LIN {X 0,Y 390.04,Z 157.401,A -85,B 0,C 180,E1 -11467.551,E2 -11467.551} C_VEL
LIN {X 0,Y 390.051,Z 157.369,A -85,B 0,C 180,E1 -11470.821,E2 -11470.821} C_VEL
LIN {X 0,Y 390.052,Z 157.382,A -85,B 0,C 180,E1 -11473.887,E2 -11473.887} C_VEL
LIN {X 0,Y 390.054,Z 157.401,A -85,B 0,C 180,E1 -11476.79,E2 -11476.79} C_VEL
LIN {X 0,Y 390.051,Z 157.386,A -85,B 0,C 180,E1 -11479.561,E2 -11479.561} C_VEL
LIN {X 0,Y 390.041,Z 157.403,A -85,B 0,C 180,E1 -11482.449,E2 -11482.449} C_VEL
LIN {X 0,Y 390.063,Z 157.38,A -85,B 0,C 180,E1 -11485.976,E2 -11485.976} C_VEL
LIN {X 0,Y 390.046,Z 157.398,A -85,B 0,C 180,E1 -11489.868,E2 -11489.868} C_VEL
LIN {X 0,Y 390.109,Z 157.374,A -85,B 0,C 180,E1 -11493.232,E2 -11493.232} C_VEL
LIN {X 0,Y 390.102,Z 157.391,A -85,B 0,C 180,E1 -11496.751,E2 -11496.751} C_VEL
LIN {X 0,Y 390.099,Z 157.374,A -85,B 0,C 180,E1 -11499.983,E2 -11499.983} C_VEL
LIN {X 0,Y 390.134,Z 157.379,A -85,B 0,C 180,E1 -11503.249,E2 -11503.249} C_VEL
LIN {X 0,Y 390.19,Z 157.377,A -85,B 0,C 180,E1 -11506.562,E2 -11506.562} C_VEL
LIN {X 0,Y 390.201,Z 157.357,A -85,B 0,C 180,E1 -11510.672,E2 -11510.672} C_VEL
LIN {X 0,Y 390.315,Z 157.357,A -85,B 0,C 180,E1 -11512.76,E2 -11512.76} C_VEL
LIN {X 0,Y 390.224,Z 157.374,A -85,B 0,C 180,E1 -11514.834,E2 -11514.834} C_VEL
LIN {X 0,Y 390.417,Z 157.337,A -85,B 0,C 180,E1 -11517.937,E2 -11517.937} C_VEL
LIN {X 0,Y 390.544,Z 157.311,A -85,B 0,C 180,E1 -11520.001,E2 -11520.001} C_VEL
LIN {X 0,Y 390.308,Z 157.36,A -85,B 0,C 180,E1 -11523.097,E2 -11523.097} C_VEL
LIN {X 0,Y 390.326,Z 157.359,A -85,B 0,C 180,E1 -11526.202,E2 -11526.202} C_VEL
LIN {X 0,Y 390.202,Z 157.354,A -85,B 0,C 180,E1 -11529.329,E2 -11529.329} C_VEL
LIN {X 0,Y 390.192,Z 157.381,A -85,B 0,C 180,E1 -11533.439,E2 -11533.439} C_VEL
LIN {X 0,Y 390.147,Z 157.369,A -85,B 0,C 180,E1 -11537.308,E2 -11537.308} C_VEL
LIN {X 0,Y 390.086,Z 157.38,A -85,B 0,C 180,E1 -11540.471,E2 -11540.471} C_VEL
LIN {X 0,Y 390.088,Z 157.392,A -85,B 0,C 180,E1 -11543.351,E2 -11543.351} C_VEL
LIN {X 0,Y 390.112,Z 157.373,A -85,B 0,C 180,E1 -11546.769,E2 -11546.769} C_VEL
LIN {X 0,Y 390.038,Z 157.398,A -85,B 0,C 180,E1 -11550.3,E2 -11550.3} C_VEL
LIN {X 0,Y 390.067,Z 157.381,A -85,B 0,C 180,E1 -11554.025,E2 -11554.025} C_VEL
LIN {X 0,Y 390.041,Z 157.398,A -85,B 0,C 180,E1 -11557.551,E2 -11557.551} C_VEL
LIN {X 0,Y 390.056,Z 157.392,A -85,B 0,C 180,E1 -11560.822,E2 -11560.822} C_VEL
LIN {X 0,Y 390.054,Z 157.396,A -85,B 0,C 180,E1 -11563.887,E2 -11563.887} C_VEL
LIN {X 0,Y 390.058,Z 157.398,A -85,B 0,C 180,E1 -11566.79,E2 -11566.79} C_VEL
LIN {X 0,Y 390.057,Z 157.377,A -85,B 0,C 180,E1 -11569.561,E2 -11569.561} C_VEL
LIN {X 0,Y 390.046,Z 157.401,A -85,B 0,C 180,E1 -11572.45,E2 -11572.45} C_VEL
LIN {X 0,Y 390.07,Z 157.396,A -85,B 0,C 180,E1 -11575.976,E2 -11575.976} C_VEL
LIN {X 0,Y 390.108,Z 157.507,A -85,B 0,C 180,E1 -11579.707,E2 -11579.707} C_VEL
LIN {X 0,Y 392.073,Z 167.322,A -85,B 0,C 180,E1 -11582.801,E2 -11582.801} C_VEL
LIN {X 0,Y 392.8,Z 173.578,A -85,B 0,C 180,E1 -11584.57,E2 -11584.57} C_VEL
LIN {X 0,Y 391.761,Z 185.813,A -85,B 0,C 180,E1 -11587.869,E2 -11587.869} C_VEL
LIN {X 0,Y 391.287,Z 191.653,A -85,B 0,C 180,E1 -11589.464,E2 -11589.464} C_VEL
LIN {X 0,Y 391.844,Z 194.823,A -85,B 0,C 180,E1 -11589.615,E2 -11589.615} C_VEL
LIN {X 0,Y 396.817,Z 222.018,A -85,B 0,C 180,E1 -11590.391,E2 -11590.391} C_VEL
LIN {X 0,Y 395.833,Z 296.555,A -85,B 0,C 180,E1 -11591.764,E2 -11591.764} C_VEL
LIN {X 0,Y 395.429,Z 307.324,A -85,B 0,C 180,E1 -11592.08,E2 -11592.08} C_VEL
LIN {X 0,Y 394.95,Z 316.424,A -85,B 0,C 180,E1 -11592.459,E2 -11592.459} C_VEL
LIN {X 0,Y 394.344,Z 326.787,A -85,B 0,C 180,E1 -11593.032,E2 -11593.032} C_VEL
LIN {X 0,Y 393.605,Z 335.919,A -85,B 0,C 180,E1 -11593.667,E2 -11593.667} C_VEL
LIN {X 0,Y 392.878,Z 344.915,A -85,B 0,C 180,E1 -11594.435,E2 -11594.435} C_VEL
LIN {X 0,Y 392.118,Z 353.643,A -85,B 0,C 180,E1 -11595.335,E2 -11595.335} C_VEL
LIN {X 0,Y 391.462,Z 361.4,A -85,B 0,C 180,E1 -11596.288,E2 -11596.288} C_VEL
LIN {X 0,Y 390.904,Z 368.261,A -85,B 0,C 180,E1 -11597.277,E2 -11597.277} C_VEL
LIN {X 0,Y 390.301,Z 374.462,A -85,B 0,C 180,E1 -11598.313,E2 -11598.313} C_VEL
LIN {X 0,Y 389.761,Z 381,A -85,B 0,C 180,E1 -11599.612,E2 -11599.612} C_VEL
LIN {X 0,Y 389.383,Z 385.501,A -85,B 0,C 180,E1 -11600.651,E2 -11600.651} C_VEL
LIN {X 0,Y 389.017,Z 390.993,A -85,B 0,C 180,E1 -11602.213,E2 -11602.213} C_VEL
LIN {X 0,Y 388.797,Z 395.317,A -85,B 0,C 180,E1 -11603.774,E2 -11603.774} C_VEL
LIN {X 0,Y 388.74,Z 397.684,A -85,B 0,C 180,E1 -11604.814,E2 -11604.814} C_VEL
LIN {X 0,Y 388.7,Z 399.482,A -85,B 0,C 180,E1 -11605.853,E2 -11605.853} C_VEL
LIN {X 0,Y 388.661,Z 401.926,A -85,B 0,C 180,E1 -11607.927,E2 -11607.927} C_VEL
LIN {X 0,Y 388.704,Z 402.515,A -85,B 0,C 180,E1 -11608.964,E2 -11608.964} C_VEL
LIN {X 0,Y 388.704,Z 402.515,A -85,B 0,C 180,E1 -11611.036,E2 -11611.036} C_VEL
LIN {X 0,Y 388.661,Z 401.926,A -85,B 0,C 180,E1 -11612.073,E2 -11612.073} C_VEL
LIN {X 0,Y 388.7,Z 399.482,A -85,B 0,C 180,E1 -11614.147,E2 -11614.147} C_VEL
LIN {X 0,Y 388.726,Z 396.43,A -85,B 0,C 180,E1 -11615.751,E2 -11615.751} C_VEL
LIN {X 0,Y 388.933,Z 392.546,A -85,B 0,C 180,E1 -11617.267,E2 -11617.267} C_VEL
LIN {X 0,Y 389.251,Z 387.417,A -85,B 0,C 180,E1 -11618.828,E2 -11618.828} C_VEL
LIN {X 0,Y 389.651,Z 382.155,A -85,B 0,C 180,E1 -11620.128,E2 -11620.128} C_VEL
LIN {X 0,Y 390.156,Z 375.837,A -85,B 0,C 180,E1 -11621.428,E2 -11621.428} C_VEL
LIN {X 0,Y 390.745,Z 369.888,A -85,B 0,C 180,E1 -11622.464,E2 -11622.464} C_VEL
LIN {X 0,Y 391.32,Z 362.959,A -85,B 0,C 180,E1 -11623.502,E2 -11623.502} C_VEL
LIN {X 0,Y 392.026,Z 354.778,A -85,B 0,C 180,E1 -11624.536,E2 -11624.536} C_VEL
LIN {X 0,Y 392.733,Z 346.266,A -85,B 0,C 180,E1 -11625.437,E2 -11625.437} C_VEL
LIN {X 0,Y 393.454,Z 337.55,A -85,B 0,C 180,E1 -11626.206,E2 -11626.206} C_VEL
LIN {X 0,Y 394.214,Z 327.793,A -85,B 0,C 180,E1 -11626.907,E2 -11626.907} C_VEL
LIN {X 0,Y 394.887,Z 317.712,A -85,B 0,C 180,E1 -11627.477,E2 -11627.477} C_VEL
LIN {X 0,Y 395.36,Z 308.197,A -85,B 0,C 180,E1 -11627.89,E2 -11627.89} C_VEL
LIN {X 0,Y 395.814,Z 297.888,A -85,B 0,C 180,E1 -11628.203,E2 -11628.203} C_VEL
LIN {X 0,Y 396.74,Z 227.164,A -85,B 0,C 180,E1 -11629.517,E2 -11629.517} C_VEL
LIN {X 0,Y 396.668,Z 221.21,A -85,B 0,C 180,E1 -11629.632,E2 -11629.632} C_VEL
LIN {X 0,Y 391.483,Z 193.035,A -85,B 0,C 180,E1 -11630.439,E2 -11630.439} C_VEL
LIN {X 0,Y 391.316,Z 191.446,A -85,B 0,C 180,E1 -11630.569,E2 -11630.569} C_VEL
LIN {X 0,Y 392.571,Z 176.893,A -85,B 0,C 180,E1 -11634.597,E2 -11634.597} C_VEL
LIN {X 0,Y 392.857,Z 172.015,A -85,B 0,C 180,E1 -11635.94,E2 -11635.94} C_VEL
LIN {X 0,Y 391.366,Z 163.735,A -85,B 0,C 180,E1 -11638.366,E2 -11638.366} C_VEL
LIN {X 0,Y 390.098,Z 157.409,A -85,B 0,C 180,E1 -11640.369,E2 -11640.369} C_VEL
LIN {X 0,Y 390.07,Z 157.397,A -85,B 0,C 180,E1 -11644.024,E2 -11644.024} C_VEL
LIN {X 0,Y 390.046,Z 157.401,A -85,B 0,C 180,E1 -11647.55,E2 -11647.55} C_VEL
LIN {X 0,Y 390.057,Z 157.379,A -85,B 0,C 180,E1 -11650.821,E2 -11650.821} C_VEL
LIN {X 0,Y 390.055,Z 157.398,A -85,B 0,C 180,E1 -11653.885,E2 -11653.885} C_VEL
LIN {X 0,Y 390.057,Z 157.396,A -85,B 0,C 180,E1 -11656.789,E2 -11656.789} C_VEL
LIN {X 0,Y 390.056,Z 157.389,A -85,B 0,C 180,E1 -11659.56,E2 -11659.56} C_VEL
LIN {X 0,Y 390.041,Z 157.398,A -85,B 0,C 180,E1 -11662.449,E2 -11662.449} C_VEL
LIN {X 0,Y 390.067,Z 157.381,A -85,B 0,C 180,E1 -11665.975,E2 -11665.975} C_VEL
LIN {X 0,Y 390.045,Z 157.396,A -85,B 0,C 180,E1 -11669.868,E2 -11669.868} C_VEL
LIN {X 0,Y 390.112,Z 157.373,A -85,B 0,C 180,E1 -11673.231,E2 -11673.231} C_VEL
LIN {X 0,Y 390.105,Z 157.391,A -85,B 0,C 180,E1 -11676.75,E2 -11676.75} C_VEL
LIN {X 0,Y 390.102,Z 157.377,A -85,B 0,C 180,E1 -11679.982,E2 -11679.982} C_VEL
LIN {X 0,Y 390.136,Z 157.379,A -85,B 0,C 180,E1 -11683.248,E2 -11683.248} C_VEL
LIN {X 0,Y 390.192,Z 157.381,A -85,B 0,C 180,E1 -11686.561,E2 -11686.561} C_VEL
LIN {X 0,Y 390.202,Z 157.354,A -85,B 0,C 180,E1 -11690.671,E2 -11690.671} C_VEL
LIN {X 0,Y 390.326,Z 157.359,A -85,B 0,C 180,E1 -11693.798,E2 -11693.798} C_VEL
LIN {X 0,Y 390.415,Z 157.346,A -85,B 0,C 180,E1 -11697.936,E2 -11697.936} C_VEL
LIN {X 0,Y 390.544,Z 157.311,A -85,B 0,C 180,E1 -11699.999,E2 -11699.999} C_VEL
LIN {X 0,Y 390.312,Z 157.36,A -85,B 0,C 180,E1 -11703.096,E2 -11703.096} C_VEL
LIN {X 0,Y 390.306,Z 157.361,A -85,B 0,C 180,E1 -11706.625,E2 -11706.625} C_VEL
LIN {X 0,Y 390.201,Z 157.357,A -85,B 0,C 180,E1 -11709.328,E2 -11709.328} C_VEL
LIN {X 0,Y 390.19,Z 157.377,A -85,B 0,C 180,E1 -11713.438,E2 -11713.438} C_VEL
LIN {X 0,Y 390.144,Z 157.379,A -85,B 0,C 180,E1 -11717.307,E2 -11717.307} C_VEL
LIN {X 0,Y 390.083,Z 157.384,A -85,B 0,C 180,E1 -11720.47,E2 -11720.47} C_VEL
LIN {X 0,Y 390.085,Z 157.394,A -85,B 0,C 180,E1 -11723.35,E2 -11723.35} C_VEL
LIN {X 0,Y 390.109,Z 157.374,A -85,B 0,C 180,E1 -11726.768,E2 -11726.768} C_VEL
LIN {X 0,Y 390.038,Z 157.399,A -85,B 0,C 180,E1 -11730.299,E2 -11730.299} C_VEL
LIN {X 0,Y 390.063,Z 157.38,A -85,B 0,C 180,E1 -11734.024,E2 -11734.024} C_VEL
LIN {X 0,Y 390.041,Z 157.403,A -85,B 0,C 180,E1 -11737.551,E2 -11737.551} C_VEL
LIN {X 0,Y 390.052,Z 157.386,A -85,B 0,C 180,E1 -11740.821,E2 -11740.821} C_VEL
LIN {X 0,Y 390.052,Z 157.396,A -85,B 0,C 180,E1 -11743.886,E2 -11743.886} C_VEL
LIN {X 0,Y 390.054,Z 157.368,A -85,B 0,C 180,E1 -11746.79,E2 -11746.79} C_VEL
LIN {X 0,Y 390.051,Z 157.377,A -85,B 0,C 180,E1 -11749.56,E2 -11749.56} C_VEL
LIN {X 0,Y 390.04,Z 157.401,A -85,B 0,C 180,E1 -11752.449,E2 -11752.449} C_VEL
LIN {X 0,Y 390.063,Z 157.376,A -85,B 0,C 180,E1 -11755.975,E2 -11755.975} C_VEL
LIN {X 0,Y 390.045,Z 157.402,A -85,B 0,C 180,E1 -11758.498,E2 -11758.498} C_VEL
LIN {X 0,Y 390.113,Z 157.387,A -85,B 0,C 180,E1 -11762.07,E2 -11762.07} C_VEL
LIN {X 0,Y 390.076,Z 157.396,A -85,B 0,C 180,E1 -11765.519,E2 -11765.519} C_VEL
LIN {X 0,Y 390.052,Z 157.401,A -85,B 0,C 180,E1 -11768.878,E2 -11768.878} C_VEL
LIN {X 0,Y 390.124,Z 157.392,A -85,B 0,C 180,E1 -11772.167,E2 -11772.167} C_VEL
LIN {X 0,Y 390.14,Z 157.389,A -85,B 0,C 180,E1 -11775.393,E2 -11775.393} C_VEL
LIN {X 0,Y 390.145,Z 157.389,A -85,B 0,C 180,E1 -11778.571,E2 -11778.571} C_VEL
LIN {X 0,Y 390.382,Z 157.657,A -85,B 0,C 180,E1 -11781.829,E2 -11781.829} C_VEL
LIN {X 0,Y 390.711,Z 158.919,A -85,B 0,C 180,E1 -11782.459,E2 -11782.459} C_VEL
LIN {X 0,Y 392.085,Z 161.236,A -85,B 0,C 180,E1 -11783.568,E2 -11783.568} C_VEL
LIN {X 0,Y 394.112,Z 162.919,A -85,B 0,C 180,E1 -11785.397,E2 -11785.397} C_VEL
LIN {X 0,Y 395.582,Z 163.492,A -85,B 0,C 180,E1 -11787.454,E2 -11787.454} C_VEL
LIN {X 0,Y 396.128,Z 163.931,A -85,B 0,C 180,E1 -11788.983,E2 -11788.983} C_VEL
LIN {X 0,Y 396.323,Z 163.848,A -85,B 0,C 180,E1 -11790,E2 -11790} C_VEL
LIN {X 0,Y 396.07,Z 163.803,A -85,B 0,C 180,E1 -11791.525,E2 -11791.525} C_VEL
LIN {X 0,Y 395.354,Z 163.371,A -85,B 0,C 180,E1 -11793.057,E2 -11793.057} C_VEL
LIN {X 0,Y 393.693,Z 162.658,A -85,B 0,C 180,E1 -11794.992,E2 -11794.992} C_VEL
LIN {X 0,Y 391.897,Z 161.019,A -85,B 0,C 180,E1 -11796.565,E2 -11796.565} C_VEL
LIN {X 0,Y 390.579,Z 158.502,A -85,B 0,C 180,E1 -11797.684,E2 -11797.684} C_VEL
LIN {X 0,Y 390.341,Z 157.593,A -85,B 0,C 180,E1 -11798.281,E2 -11798.281} C_VEL
LIN {X 0,Y 390.145,Z 157.389,A -85,B 0,C 180,E1 -11801.429,E2 -11801.429} C_VEL
LIN {X 0,Y 390.14,Z 157.39,A -85,B 0,C 180,E1 -11804.607,E2 -11804.607} C_VEL
LIN {X 0,Y 390.124,Z 157.392,A -85,B 0,C 180,E1 -11807.833,E2 -11807.833} C_VEL
LIN {X 0,Y 390.052,Z 157.401,A -85,B 0,C 180,E1 -11811.122,E2 -11811.122} C_VEL
LIN {X 0,Y 390.076,Z 157.396,A -85,B 0,C 180,E1 -11814.481,E2 -11814.481} C_VEL
LIN {X 0,Y 390.111,Z 157.387,A -85,B 0,C 180,E1 -11818.025,E2 -11818.025} C_VEL
LIN {X 0,Y 390.022,Z 157.396,A -85,B 0,C 180,E1 -11820.799,E2 -11820.799} C_VEL
LIN {X 0,Y 389.356,Z 157.487,A -85,B 0,C 180,E1 -11821.661,E2 -11821.661} C_VEL
LIN {X 0,Y 386.503,Z 157.831,A -85,B 0,C 180,E1 -11823.063,E2 -11823.063} C_VEL
LIN {X 0,Y 384.095,Z 158.119,A -85,B 0,C 180,E1 -11824.195,E2 -11824.195} C_VEL
LIN {X 0,Y 383.071,Z 158.245,A -85,B 0,C 180,E1 -11825.071,E2 -11825.071} C_VEL
LIN {X 0,Y 382.994,Z 158.257,A -85,B 0,C 180,E1 -11825.368,E2 -11825.368} C_VEL
LIN {X 0,Y 383.001,Z 158.279,A -85,B 0,C 180,E1 -11828.601,E2 -11828.601} C_VEL
LIN {X 0,Y 382.978,Z 158.243,A -85,B 0,C 180,E1 -11831.348,E2 -11831.348} C_VEL
LIN {X 0,Y 382.994,Z 158.262,A -85,B 0,C 180,E1 -11834.304,E2 -11834.304} C_VEL
LIN {X 0,Y 383.005,Z 158.274,A -85,B 0,C 180,E1 -11837.24,E2 -11837.24} C_VEL
LIN {X 0,Y 383.011,Z 158.267,A -85,B 0,C 180,E1 -11840.414,E2 -11840.414} C_VEL
LIN {X 0,Y 383.022,Z 158.271,A -85,B 0,C 180,E1 -11844.045,E2 -11844.045} C_VEL
LIN {X 0,Y 382.983,Z 158.274,A -85,B 0,C 180,E1 -11847.578,E2 -11847.578} C_VEL
LIN {X 0,Y 382.992,Z 158.275,A -85,B 0,C 180,E1 -11850.301,E2 -11850.301} C_VEL
LIN {X 0,Y 383.052,Z 158.251,A -85,B 0,C 180,E1 -11852.698,E2 -11852.698} C_VEL
LIN {X 0,Y 383.048,Z 158.266,A -85,B 0,C 180,E1 -11855.04,E2 -11855.04} C_VEL
LIN {X 0,Y 382.989,Z 158.271,A -85,B 0,C 180,E1 -11858.469,E2 -11858.469} C_VEL
LIN {X 0,Y 383.058,Z 158.247,A -85,B 0,C 180,E1 -11861.827,E2 -11861.827} C_VEL
LIN {X 0,Y 383.106,Z 158.261,A -85,B 0,C 180,E1 -11865.119,E2 -11865.119} C_VEL
LIN {X 0,Y 383.093,Z 158.249,A -85,B 0,C 180,E1 -11868.358,E2 -11868.358} C_VEL
LIN {X 0,Y 383.3,Z 158.225,A -85,B 0,C 180,E1 -11871.933,E2 -11871.933} C_VEL
LIN {X 0,Y 383.196,Z 158.25,A -85,B 0,C 180,E1 -11874.739,E2 -11874.739} C_VEL
LIN {X 0,Y 383.384,Z 158.213,A -85,B 0,C 180,E1 -11877.899,E2 -11877.899} C_VEL
LIN {X 0,Y 383.514,Z 158.186,A -85,B 0,C 180,E1 -11880.001,E2 -11880.001} C_VEL
LIN {X 0,Y 383.244,Z 158.24,A -85,B 0,C 180,E1 -11883.154,E2 -11883.154} C_VEL
LIN {X 0,Y 383.282,Z 158.236,A -85,B 0,C 180,E1 -11886.317,E2 -11886.317} C_VEL
LIN {X 0,Y 383.148,Z 158.231,A -85,B 0,C 180,E1 -11889.503,E2 -11889.503} C_VEL
LIN {X 0,Y 383.123,Z 158.261,A -85,B 0,C 180,E1 -11893.537,E2 -11893.537} C_VEL
LIN {X 0,Y 383.092,Z 158.245,A -85,B 0,C 180,E1 -11897.455,E2 -11897.455} C_VEL
LIN {X 0,Y 383.029,Z 158.26,A -85,B 0,C 180,E1 -11900.649,E2 -11900.649} C_VEL
LIN {X 0,Y 383.032,Z 158.268,A -85,B 0,C 180,E1 -11903.808,E2 -11903.808} C_VEL
LIN {X 0,Y 383.055,Z 158.252,A -85,B 0,C 180,E1 -11907.303,E2 -11907.303} C_VEL
LIN {X 0,Y 382.982,Z 158.281,A -85,B 0,C 180,E1 -11910.919,E2 -11910.919} C_VEL
LIN {X 0,Y 383.017,Z 158.26,A -85,B 0,C 180,E1 -11914.669,E2 -11914.669} C_VEL
LIN {X 0,Y 382.997,Z 158.276,A -85,B 0,C 180,E1 -11917.904,E2 -11917.904} C_VEL
LIN {X 0,Y 382.983,Z 158.275,A -85,B 0,C 180,E1 -11921.348,E2 -11921.348} C_VEL
LIN {X 0,Y 382.996,Z 158.273,A -85,B 0,C 180,E1 -11924.304,E2 -11924.304} C_VEL
LIN {X 0,Y 383.011,Z 158.274,A -85,B 0,C 180,E1 -11927.241,E2 -11927.241} C_VEL
LIN {X 0,Y 383.017,Z 158.257,A -85,B 0,C 180,E1 -11930.414,E2 -11930.414} C_VEL
LIN {X 0,Y 383.027,Z 158.262,A -85,B 0,C 180,E1 -11934.045,E2 -11934.045} C_VEL
LIN {X 0,Y 382.988,Z 158.271,A -85,B 0,C 180,E1 -11937.579,E2 -11937.579} C_VEL
LIN {X 0,Y 383.085,Z 158.439,A -85,B 0,C 180,E1 -11939.428,E2 -11939.428} C_VEL
LIN {X 0,Y 385.219,Z 169.231,A -85,B 0,C 180,E1 -11942.864,E2 -11942.864} C_VEL
LIN {X 0,Y 385.823,Z 174.445,A -85,B 0,C 180,E1 -11944.366,E2 -11944.366} C_VEL
LIN {X 0,Y 384.863,Z 185.625,A -85,B 0,C 180,E1 -11947.451,E2 -11947.451} C_VEL
LIN {X 0,Y 384.402,Z 191.46,A -85,B 0,C 180,E1 -11949.078,E2 -11949.078} C_VEL
LIN {X 0,Y 384.807,Z 194.101,A -85,B 0,C 180,E1 -11949.215,E2 -11949.215} C_VEL
LIN {X 0,Y 389.909,Z 221.418,A -85,B 0,C 180,E1 -11950.021,E2 -11950.021} C_VEL
LIN {X 0,Y 390.122,Z 228.726,A -85,B 0,C 180,E1 -11950.172,E2 -11950.172} C_VEL
LIN {X 0,Y 389.1,Z 296.364,A -85,B 0,C 180,E1 -11951.437,E2 -11951.437} C_VEL
LIN {X 0,Y 388.692,Z 307.133,A -85,B 0,C 180,E1 -11951.758,E2 -11951.758} C_VEL
LIN {X 0,Y 388.187,Z 316.232,A -85,B 0,C 180,E1 -11952.143,E2 -11952.143} C_VEL
LIN {X 0,Y 387.553,Z 326.595,A -85,B 0,C 180,E1 -11952.726,E2 -11952.726} C_VEL
LIN {X 0,Y 386.785,Z 335.727,A -85,B 0,C 180,E1 -11953.371,E2 -11953.371} C_VEL
LIN {X 0,Y 386.013,Z 344.723,A -85,B 0,C 180,E1 -11954.151,E2 -11954.151} C_VEL
LIN {X 0,Y 385.217,Z 353.451,A -85,B 0,C 180,E1 -11955.067,E2 -11955.067} C_VEL
LIN {X 0,Y 384.53,Z 361.407,A -85,B 0,C 180,E1 -11956.064,E2 -11956.064} C_VEL
LIN {X 0,Y 383.793,Z 369.696,A -85,B 0,C 180,E1 -11957.306,E2 -11957.306} C_VEL
LIN {X 0,Y 383.174,Z 375.645,A -85,B 0,C 180,E1 -11958.36,E2 -11958.36} C_VEL
LIN {X 0,Y 382.642,Z 381.963,A -85,B 0,C 180,E1 -11959.684,E2 -11959.684} C_VEL
LIN {X 0,Y 382.207,Z 387.225,A -85,B 0,C 180,E1 -11961.008,E2 -11961.008} C_VEL
LIN {X 0,Y 381.861,Z 392.354,A -85,B 0,C 180,E1 -11962.598,E2 -11962.598} C_VEL
LIN {X 0,Y 381.688,Z 395.641,A -85,B 0,C 180,E1 -11963.883,E2 -11963.883} C_VEL
LIN {X 0,Y 381.641,Z 397.491,A -85,B 0,C 180,E1 -11964.717,E2 -11964.717} C_VEL
LIN {X 0,Y 381.625,Z 399.291,A -85,B 0,C 180,E1 -11965.776,E2 -11965.776} C_VEL
LIN {X 0,Y 381.56,Z 401.734,A -85,B 0,C 180,E1 -11967.889,E2 -11967.889} C_VEL
LIN {X 0,Y 381.604,Z 402.323,A -85,B 0,C 180,E1 -11968.945,E2 -11968.945} C_VEL
LIN {X 0,Y 381.604,Z 402.323,A -85,B 0,C 180,E1 -11971.055,E2 -11971.055} C_VEL
LIN {X 0,Y 381.56,Z 401.734,A -85,B 0,C 180,E1 -11972.111,E2 -11972.111} C_VEL
LIN {X 0,Y 381.625,Z 399.291,A -85,B 0,C 180,E1 -11974.224,E2 -11974.224} C_VEL
LIN {X 0,Y 381.64,Z 397.491,A -85,B 0,C 180,E1 -11975.283,E2 -11975.283} C_VEL
LIN {X 0,Y 381.781,Z 393.884,A -85,B 0,C 180,E1 -11976.872,E2 -11976.872} C_VEL
LIN {X 0,Y 382.058,Z 389.14,A -85,B 0,C 180,E1 -11978.462,E2 -11978.462} C_VEL
LIN {X 0,Y 382.525,Z 383.118,A -85,B 0,C 180,E1 -11980.052,E2 -11980.052} C_VEL
LIN {X 0,Y 383.053,Z 377.021,A -85,B 0,C 180,E1 -11981.375,E2 -11981.375} C_VEL
LIN {X 0,Y 383.643,Z 371.322,A -85,B 0,C 180,E1 -11982.43,E2 -11982.43} C_VEL
LIN {X 0,Y 384.369,Z 362.766,A -85,B 0,C 180,E1 -11983.751,E2 -11983.751} C_VEL
LIN {X 0,Y 385.145,Z 354.586,A -85,B 0,C 180,E1 -11984.801,E2 -11984.801} C_VEL
LIN {X 0,Y 385.892,Z 346.074,A -85,B 0,C 180,E1 -11985.718,E2 -11985.718} C_VEL
LIN {X 0,Y 386.646,Z 337.359,A -85,B 0,C 180,E1 -11986.5,E2 -11986.5} C_VEL
LIN {X 0,Y 387.424,Z 327.601,A -85,B 0,C 180,E1 -11987.212,E2 -11987.212} C_VEL
LIN {X 0,Y 388.107,Z 317.52,A -85,B 0,C 180,E1 -11987.793,E2 -11987.793} C_VEL
LIN {X 0,Y 388.626,Z 308.006,A -85,B 0,C 180,E1 -11988.211,E2 -11988.211} C_VEL
LIN {X 0,Y 389.083,Z 297.696,A -85,B 0,C 180,E1 -11988.529,E2 -11988.529} C_VEL
LIN {X 0,Y 390.038,Z 230.896,A -85,B 0,C 180,E1 -11989.791,E2 -11989.791} C_VEL
LIN {X 0,Y 389.98,Z 222.068,A -85,B 0,C 180,E1 -11989.963,E2 -11989.963} C_VEL
LIN {X 0,Y 384.819,Z 193.984,A -85,B 0,C 180,E1 -11990.787,E2 -11990.787} C_VEL
LIN {X 0,Y 384.39,Z 191.454,A -85,B 0,C 180,E1 -11990.923,E2 -11990.923} C_VEL
LIN {X 0,Y 385.748,Z 176.712,A -85,B 0,C 180,E1 -11995.061,E2 -11995.061} C_VEL
LIN {X 0,Y 385.917,Z 173.701,A -85,B 0,C 180,E1 -11995.917,E2 -11995.917} C_VEL
LIN {X 0,Y 384.497,Z 165.445,A -85,B 0,C 180,E1 -11998.375,E2 -11998.375} C_VEL
LIN {X 0,Y 383.049,Z 158.304,A -85,B 0,C 180,E1 -12000.653,E2 -12000.653} C_VEL
LIN {X 0,Y 383.019,Z 158.268,A -85,B 0,C 180,E1 -12004.667,E2 -12004.667} C_VEL
LIN {X 0,Y 383.002,Z 158.277,A -85,B 0,C 180,E1 -12007.903,E2 -12007.903} C_VEL
LIN {X 0,Y 382.984,Z 158.263,A -85,B 0,C 180,E1 -12011.347,E2 -12011.347} C_VEL
LIN {X 0,Y 382.996,Z 158.274,A -85,B 0,C 180,E1 -12014.303,E2 -12014.303} C_VEL
LIN {X 0,Y 383.01,Z 158.277,A -85,B 0,C 180,E1 -12017.24,E2 -12017.24} C_VEL
LIN {X 0,Y 383.013,Z 158.265,A -85,B 0,C 180,E1 -12020.413,E2 -12020.413} C_VEL
LIN {X 0,Y 383.024,Z 158.267,A -85,B 0,C 180,E1 -12024.044,E2 -12024.044} C_VEL
LIN {X 0,Y 382.986,Z 158.275,A -85,B 0,C 180,E1 -12027.577,E2 -12027.577} C_VEL
LIN {X 0,Y 382.991,Z 158.275,A -85,B 0,C 180,E1 -12030.299,E2 -12030.299} C_VEL
LIN {X 0,Y 383.079,Z 158.252,A -85,B 0,C 180,E1 -12034.02,E2 -12034.02} C_VEL
LIN {X 0,Y 383.011,Z 158.273,A -85,B 0,C 180,E1 -12037.335,E2 -12037.335} C_VEL
LIN {X 0,Y 383.058,Z 158.247,A -85,B 0,C 180,E1 -12040.716,E2 -12040.716} C_VEL
LIN {X 0,Y 383.078,Z 158.258,A -85,B 0,C 180,E1 -12044.026,E2 -12044.026} C_VEL
LIN {X 0,Y 383.134,Z 158.252,A -85,B 0,C 180,E1 -12047.283,E2 -12047.283} C_VEL
LIN {X 0,Y 383.148,Z 158.231,A -85,B 0,C 180,E1 -12050.497,E2 -12050.497} C_VEL
LIN {X 0,Y 383.282,Z 158.236,A -85,B 0,C 180,E1 -12053.683,E2 -12053.683} C_VEL
LIN {X 0,Y 383.382,Z 158.222,A -85,B 0,C 180,E1 -12057.898,E2 -12057.898} C_VEL
LIN {X 0,Y 383.514,Z 158.186,A -85,B 0,C 180,E1 -12059.999,E2 -12059.999} C_VEL
LIN {X 0,Y 383.248,Z 158.239,A -85,B 0,C 180,E1 -12063.153,E2 -12063.153} C_VEL
LIN {X 0,Y 383.266,Z 158.238,A -85,B 0,C 180,E1 -12066.618,E2 -12066.618} C_VEL
LIN {X 0,Y 383.256,Z 158.225,A -85,B 0,C 180,E1 -12068.435,E2 -12068.435} C_VEL
LIN {X 0,Y 383.093,Z 158.249,A -85,B 0,C 180,E1 -12071.642,E2 -12071.642} C_VEL
LIN {X 0,Y 383.106,Z 158.261,A -85,B 0,C 180,E1 -12074.881,E2 -12074.881} C_VEL
LIN {X 0,Y 383.058,Z 158.247,A -85,B 0,C 180,E1 -12078.173,E2 -12078.173} C_VEL
LIN {X 0,Y 382.989,Z 158.271,A -85,B 0,C 180,E1 -12081.531,E2 -12081.531} C_VEL
LIN {X 0,Y 383.048,Z 158.266,A -85,B 0,C 180,E1 -12084.96,E2 -12084.96} C_VEL
LIN {X 0,Y 383.044,Z 158.261,A -85,B 0,C 180,E1 -12088.492,E2 -12088.492} C_VEL
LIN {X 0,Y 383.006,Z 158.272,A -85,B 0,C 180,E1 -12092.149,E2 -12092.149} C_VEL
LIN {X 0,Y 383.013,Z 158.256,A -85,B 0,C 180,E1 -12094.668,E2 -12094.668} C_VEL
LIN {X 0,Y 382.997,Z 158.277,A -85,B 0,C 180,E1 -12097.904,E2 -12097.904} C_VEL
LIN {X 0,Y 382.98,Z 158.27,A -85,B 0,C 180,E1 -12101.347,E2 -12101.347} C_VEL
LIN {X 0,Y 382.994,Z 158.274,A -85,B 0,C 180,E1 -12104.304,E2 -12104.304} C_VEL
LIN {X 0,Y 383.005,Z 158.239,A -85,B 0,C 180,E1 -12107.24,E2 -12107.24} C_VEL
LIN {X 0,Y 383.01,Z 158.266,A -85,B 0,C 180,E1 -12110.413,E2 -12110.413} C_VEL
LIN {X 0,Y 383.022,Z 158.262,A -85,B 0,C 180,E1 -12114.045,E2 -12114.045} C_VEL
LIN {X 0,Y 383.033,Z 158.272,A -85,B 0,C 180,E1 -12117.853,E2 -12117.853} C_VEL
LIN {X 0,Y 383.059,Z 158.261,A -85,B 0,C 180,E1 -12121.72,E2 -12121.72} C_VEL
LIN {X 0,Y 383.048,Z 158.273,A -85,B 0,C 180,E1 -12125.04,E2 -12125.04} C_VEL
LIN {X 0,Y 382.989,Z 158.281,A -85,B 0,C 180,E1 -12128.469,E2 -12128.469} C_VEL
LIN {X 0,Y 383.085,Z 158.268,A -85,B 0,C 180,E1 -12131.828,E2 -12131.828} C_VEL
LIN {X 0,Y 383.106,Z 158.266,A -85,B 0,C 180,E1 -12135.118,E2 -12135.118} C_VEL
LIN {X 0,Y 383.113,Z 158.39,A -85,B 0,C 180,E1 -12138.359,E2 -12138.359} C_VEL
LIN {X 0,Y 383.303,Z 159.256,A -85,B 0,C 180,E1 -12138.867,E2 -12138.867} C_VEL
LIN {X 0,Y 384.444,Z 161.599,A -85,B 0,C 180,E1 -12139.533,E2 -12139.533} C_VEL
LIN {X 0,Y 386.582,Z 163.495,A -85,B 0,C 180,E1 -12140.583,E2 -12140.583} C_VEL
LIN {X 0,Y 388.921,Z 164.829,A -85,B 0,C 180,E1 -12141.896,E2 -12141.896} C_VEL
LIN {X 0,Y 390.34,Z 167.396,A -85,B 0,C 180,E1 -12142.955,E2 -12142.955} C_VEL
LIN {X 0,Y 391.933,Z 169.071,A -85,B 0,C 180,E1 -12144.211,E2 -12144.211} C_VEL
LIN {X 0,Y 393.437,Z 170.033,A -85,B 0,C 180,E1 -12145.646,E2 -12145.646} C_VEL
LIN {X 0,Y 394.719,Z 170.512,A -85,B 0,C 180,E1 -12147.449,E2 -12147.449} C_VEL
LIN {X 0,Y 395.266,Z 170.977,A -85,B 0,C 180,E1 -12148.981,E2 -12148.981} C_VEL
LIN {X 0,Y 395.458,Z 170.896,A -85,B 0,C 180,E1 -12150,E2 -12150} C_VEL
LIN {X 0,Y 395.202,Z 170.852,A -85,B 0,C 180,E1 -12151.529,E2 -12151.529} C_VEL
LIN {X 0,Y 394.244,Z 170.355,A -85,B 0,C 180,E1 -12153.368,E2 -12153.368} C_VEL
LIN {X 0,Y 392.65,Z 169.62,A -85,B 0,C 180,E1 -12155.134,E2 -12155.134} C_VEL
LIN {X 0,Y 390.787,Z 167.978,A -85,B 0,C 180,E1 -12156.713,E2 -12156.713} C_VEL
LIN {X 0,Y 389.246,Z 165.411,A -85,B 0,C 180,E1 -12157.901,E2 -12157.901} C_VEL
LIN {X 0,Y 388.306,Z 164.316,A -85,B 0,C 180,E1 -12158.456,E2 -12158.456} C_VEL
LIN {X 0,Y 385.837,Z 163.007,A -85,B 0,C 180,E1 -12159.766,E2 -12159.766} C_VEL
LIN {X 0,Y 383.934,Z 160.79,A -85,B 0,C 180,E1 -12160.748,E2 -12160.748} C_VEL
LIN {X 0,Y 383.222,Z 158.963,A -85,B 0,C 180,E1 -12161.236,E2 -12161.236} C_VEL
LIN {X 0,Y 383.115,Z 158.297,A -85,B 0,C 180,E1 -12161.91,E2 -12161.91} C_VEL
LIN {X 0,Y 383.106,Z 158.266,A -85,B 0,C 180,E1 -12164.882,E2 -12164.882} C_VEL
LIN {X 0,Y 383.085,Z 158.268,A -85,B 0,C 180,E1 -12168.172,E2 -12168.172} C_VEL
LIN {X 0,Y 382.989,Z 158.281,A -85,B 0,C 180,E1 -12171.531,E2 -12171.531} C_VEL
LIN {X 0,Y 383.048,Z 158.273,A -85,B 0,C 180,E1 -12174.96,E2 -12174.96} C_VEL
LIN {X 0,Y 383.045,Z 158.26,A -85,B 0,C 180,E1 -12178.492,E2 -12178.492} C_VEL
LIN {X 0,Y 383.023,Z 158.274,A -85,B 0,C 180,E1 -12182.432,E2 -12182.432} C_VEL
LIN {X 0,Y 382.994,Z 158.257,A -85,B 0,C 180,E1 -12185.368,E2 -12185.368} C_VEL
LIN {X 0,Y 382.357,Z 158.348,A -85,B 0,C 180,E1 -12186.246,E2 -12186.246} C_VEL
LIN {X 0,Y 379.562,Z 158.711,A -85,B 0,C 180,E1 -12187.674,E2 -12187.674} C_VEL
LIN {X 0,Y 377.157,Z 159.01,A -85,B 0,C 180,E1 -12188.828,E2 -12188.828} C_VEL
LIN {X 0,Y 376.086,Z 159.131,A -85,B 0,C 180,E1 -12189.72,E2 -12189.72} C_VEL
LIN {X 0,Y 375.978,Z 159.137,A -85,B 0,C 180,E1 -12190.022,E2 -12190.022} C_VEL
LIN {X 0,Y 375.927,Z 159.136,A -85,B 0,C 180,E1 -12193.766,E2 -12193.766} C_VEL
LIN {X 0,Y 375.93,Z 159.16,A -85,B 0,C 180,E1 -12196.811,E2 -12196.811} C_VEL
LIN {X 0,Y 375.959,Z 159.146,A -85,B 0,C 180,E1 -12200.538,E2 -12200.538} C_VEL
LIN {X 0,Y 375.96,Z 159.15,A -85,B 0,C 180,E1 -12203.496,E2 -12203.496} C_VEL
LIN {X 0,Y 375.955,Z 159.136,A -85,B 0,C 180,E1 -12205.889,E2 -12205.889} C_VEL
LIN {X 0,Y 375.963,Z 159.152,A -85,B 0,C 180,E1 -12209.688,E2 -12209.688} C_VEL
LIN {X 0,Y 375.997,Z 159.132,A -85,B 0,C 180,E1 -12212.142,E2 -12212.142} C_VEL
LIN {X 0,Y 376.002,Z 159.141,A -85,B 0,C 180,E1 -12214.539,E2 -12214.539} C_VEL
LIN {X 0,Y 375.959,Z 159.152,A -85,B 0,C 180,E1 -12218.046,E2 -12218.046} C_VEL
LIN {X 0,Y 376.004,Z 159.122,A -85,B 0,C 180,E1 -12221.474,E2 -12221.474} C_VEL
LIN {X 0,Y 376.054,Z 159.14,A -85,B 0,C 180,E1 -12224.833,E2 -12224.833} C_VEL
LIN {X 0,Y 376.045,Z 159.129,A -85,B 0,C 180,E1 -12228.137,E2 -12228.137} C_VEL
LIN {X 0,Y 376.254,Z 159.101,A -85,B 0,C 180,E1 -12231.878,E2 -12231.878} C_VEL
LIN {X 0,Y 376.168,Z 159.125,A -85,B 0,C 180,E1 -12234.64,E2 -12234.64} C_VEL
LIN {X 0,Y 376.35,Z 159.089,A -85,B 0,C 180,E1 -12237.86,E2 -12237.86} C_VEL
LIN {X 0,Y 376.483,Z 159.061,A -85,B 0,C 180,E1 -12240.001,E2 -12240.001} C_VEL
LIN {X 0,Y 376.183,Z 159.121,A -85,B 0,C 180,E1 -12243.214,E2 -12243.214} C_VEL
LIN {X 0,Y 376.24,Z 159.113,A -85,B 0,C 180,E1 -12246.436,E2 -12246.436} C_VEL
LIN {X 0,Y 376.116,Z 159.106,A -85,B 0,C 180,E1 -12249.682,E2 -12249.682} C_VEL
LIN {X 0,Y 376.087,Z 159.136,A -85,B 0,C 180,E1 -12253.658,E2 -12253.658} C_VEL
LIN {X 0,Y 376.041,Z 159.121,A -85,B 0,C 180,E1 -12257.607,E2 -12257.607} C_VEL
LIN {X 0,Y 375.976,Z 159.14,A -85,B 0,C 180,E1 -12260.833,E2 -12260.833} C_VEL
LIN {X 0,Y 375.992,Z 159.145,A -85,B 0,C 180,E1 -12264.282,E2 -12264.282} C_VEL
LIN {X 0,Y 376.018,Z 159.127,A -85,B 0,C 180,E1 -12266.653,E2 -12266.653} C_VEL
LIN {X 0,Y 375.964,Z 159.152,A -85,B 0,C 180,E1 -12270.313,E2 -12270.313} C_VEL
LIN {X 0,Y 375.959,Z 159.137,A -85,B 0,C 180,E1 -12274.112,E2 -12274.112} C_VEL
LIN {X 0,Y 375.952,Z 159.156,A -85,B 0,C 180,E1 -12276.742,E2 -12276.742} C_VEL
LIN {X 0,Y 375.987,Z 159.14,A -85,B 0,C 180,E1 -12279.971,E2 -12279.971} C_VEL
LIN {X 0,Y 375.93,Z 159.155,A -85,B 0,C 180,E1 -12283.767,E2 -12283.767} C_VEL
LIN {X 0,Y 375.935,Z 159.157,A -85,B 0,C 180,E1 -12286.811,E2 -12286.811} C_VEL
LIN {X 0,Y 375.964,Z 159.136,A -85,B 0,C 180,E1 -12290.538,E2 -12290.538} C_VEL
LIN {X 0,Y 375.966,Z 159.147,A -85,B 0,C 180,E1 -12293.496,E2 -12293.496} C_VEL
LIN {X 0,Y 375.962,Z 159.152,A -85,B 0,C 180,E1 -12295.889,E2 -12295.889} C_VEL
LIN {X 0,Y 375.988,Z 159.295,A -85,B 0,C 180,E1 -12299.095,E2 -12299.095} C_VEL
LIN {X 0,Y 377.978,Z 169.05,A -85,B 0,C 180,E1 -12302.3,E2 -12302.3} C_VEL
LIN {X 0,Y 378.867,Z 175.313,A -85,B 0,C 180,E1 -12304.156,E2 -12304.156} C_VEL
LIN {X 0,Y 377.992,Z 185.438,A -85,B 0,C 180,E1 -12307.018,E2 -12307.018} C_VEL
LIN {X 0,Y 377.482,Z 191.342,A -85,B 0,C 180,E1 -12308.688,E2 -12308.688} C_VEL
LIN {X 0,Y 378.456,Z 196.459,A -85,B 0,C 180,E1 -12308.9,E2 -12308.9} C_VEL
LIN {X 0,Y 383.326,Z 222.881,A -85,B 0,C 180,E1 -12309.695,E2 -12309.695} C_VEL
LIN {X 0,Y 383.032,Z 254.972,A -85,B 0,C 180,E1 -12310.305,E2 -12310.305} C_VEL
LIN {X 0,Y 382.334,Z 297.504,A -85,B 0,C 180,E1 -12311.131,E2 -12311.131} C_VEL
LIN {X 0,Y 381.921,Z 307.815,A -85,B 0,C 180,E1 -12311.458,E2 -12311.458} C_VEL
LIN {X 0,Y 381.355,Z 317.328,A -85,B 0,C 180,E1 -12311.881,E2 -12311.881} C_VEL
LIN {X 0,Y 380.707,Z 327.411,A -85,B 0,C 180,E1 -12312.474,E2 -12312.474} C_VEL
LIN {X 0,Y 379.85,Z 337.167,A -85,B 0,C 180,E1 -12313.196,E2 -12313.196} C_VEL
LIN {X 0,Y 378.925,Z 347.234,A -85,B 0,C 180,E1 -12314.123,E2 -12314.123} C_VEL
LIN {X 0,Y 377.876,Z 358.621,A -85,B 0,C 180,E1 -12315.442,E2 -12315.442} C_VEL
LIN {X 0,Y 377.032,Z 367.877,A -85,B 0,C 180,E1 -12316.801,E2 -12316.801} C_VEL
LIN {X 0,Y 376.374,Z 374.078,A -85,B 0,C 180,E1 -12317.874,E2 -12317.874} C_VEL
LIN {X 0,Y 375.696,Z 380.614,A -85,B 0,C 180,E1 -12319.219,E2 -12319.219} C_VEL
LIN {X 0,Y 375.324,Z 385.116,A -85,B 0,C 180,E1 -12320.298,E2 -12320.298} C_VEL
LIN {X 0,Y 374.882,Z 390.607,A -85,B 0,C 180,E1 -12321.917,E2 -12321.917} C_VEL
LIN {X 0,Y 374.633,Z 394.932,A -85,B 0,C 180,E1 -12323.537,E2 -12323.537} C_VEL
LIN {X 0,Y 374.551,Z 397.299,A -85,B 0,C 180,E1 -12324.617,E2 -12324.617} C_VEL
LIN {X 0,Y 374.529,Z 399.099,A -85,B 0,C 180,E1 -12325.695,E2 -12325.695} C_VEL
LIN {X 0,Y 374.459,Z 401.542,A -85,B 0,C 180,E1 -12327.849,E2 -12327.849} C_VEL
LIN {X 0,Y 374.504,Z 402.132,A -85,B 0,C 180,E1 -12328.925,E2 -12328.925} C_VEL
LIN {X 0,Y 374.504,Z 402.132,A -85,B 0,C 180,E1 -12331.075,E2 -12331.075} C_VEL
LIN {X 0,Y 374.459,Z 401.542,A -85,B 0,C 180,E1 -12332.151,E2 -12332.151} C_VEL
LIN {X 0,Y 374.529,Z 399.098,A -85,B 0,C 180,E1 -12334.305,E2 -12334.305} C_VEL
LIN {X 0,Y 374.583,Z 395.831,A -85,B 0,C 180,E1 -12336.064,E2 -12336.064} C_VEL
LIN {X 0,Y 374.794,Z 392.162,A -85,B 0,C 180,E1 -12337.542,E2 -12337.542} C_VEL
LIN {X 0,Y 375.163,Z 387.032,A -85,B 0,C 180,E1 -12339.162,E2 -12339.162} C_VEL
LIN {X 0,Y 375.626,Z 381.77,A -85,B 0,C 180,E1 -12340.511,E2 -12340.511} C_VEL
LIN {X 0,Y 376.203,Z 375.453,A -85,B 0,C 180,E1 -12341.858,E2 -12341.858} C_VEL
LIN {X 0,Y 376.864,Z 369.504,A -85,B 0,C 180,E1 -12342.931,E2 -12342.931} C_VEL
LIN {X 0,Y 377.596,Z 361.36,A -85,B 0,C 180,E1 -12344.176,E2 -12344.176} C_VEL
LIN {X 0,Y 378.496,Z 352.125,A -85,B 0,C 180,E1 -12345.343,E2 -12345.343} C_VEL
LIN {X 0,Y 379.437,Z 341.828,A -85,B 0,C 180,E1 -12346.407,E2 -12346.407} C_VEL
LIN {X 0,Y 380.5,Z 329.423,A -85,B 0,C 180,E1 -12347.397,E2 -12347.397} C_VEL
LIN {X 0,Y 381.298,Z 318.617,A -85,B 0,C 180,E1 -12348.052,E2 -12348.052} C_VEL
LIN {X 0,Y 381.847,Z 308.689,A -85,B 0,C 180,E1 -12348.511,E2 -12348.511} C_VEL
LIN {X 0,Y 382.337,Z 298.837,A -85,B 0,C 180,E1 -12348.834,E2 -12348.834} C_VEL
LIN {X 0,Y 382.804,Z 274.614,A -85,B 0,C 180,E1 -12349.324,E2 -12349.324} C_VEL
LIN {X 0,Y 383.354,Z 223.195,A -85,B 0,C 180,E1 -12350.297,E2 -12350.297} C_VEL
LIN {X 0,Y 378.048,Z 194.446,A -85,B 0,C 180,E1 -12351.164,E2 -12351.164} C_VEL
LIN {X 0,Y 377.471,Z 191.356,A -85,B 0,C 180,E1 -12351.308,E2 -12351.308} C_VEL
LIN {X 0,Y 378.946,Z 176.531,A -85,B 0,C 180,E1 -12355.543,E2 -12355.543} C_VEL
LIN {X 0,Y 378.518,Z 171.762,A -85,B 0,C 180,E1 -12356.972,E2 -12356.972} C_VEL
LIN {X 0,Y 376.396,Z 161.131,A -85,B 0,C 180,E1 -12360.274,E2 -12360.274} C_VEL
LIN {X 0,Y 375.977,Z 159.205,A -85,B 0,C 180,E1 -12360.965,E2 -12360.965} C_VEL
LIN {X 0,Y 375.981,Z 159.144,A -85,B 0,C 180,E1 -12364.667,E2 -12364.667} C_VEL
LIN {X 0,Y 375.977,Z 159.149,A -85,B 0,C 180,E1 -12368.27,E2 -12368.27} C_VEL
LIN {X 0,Y 375.935,Z 159.144,A -85,B 0,C 180,E1 -12371.6,E2 -12371.6} C_VEL
LIN {X 0,Y 375.927,Z 159.152,A -85,B 0,C 180,E1 -12375.268,E2 -12375.268} C_VEL
LIN {X 0,Y 375.934,Z 159.154,A -85,B 0,C 180,E1 -12378.399,E2 -12378.399} C_VEL
LIN {X 0,Y 375.972,Z 159.153,A -85,B 0,C 180,E1 -12381.729,E2 -12381.729} C_VEL
LIN {X 0,Y 375.979,Z 159.137,A -85,B 0,C 180,E1 -12385.332,E2 -12385.332} C_VEL
LIN {X 0,Y 375.957,Z 159.151,A -85,B 0,C 180,E1 -12388.437,E2 -12388.437} C_VEL
LIN {X 0,Y 375.982,Z 159.136,A -85,B 0,C 180,E1 -12392.14,E2 -12392.14} C_VEL
LIN {X 0,Y 376.005,Z 159.134,A -85,B 0,C 180,E1 -12394.538,E2 -12394.538} C_VEL
LIN {X 0,Y 375.966,Z 159.148,A -85,B 0,C 180,E1 -12398.045,E2 -12398.045} C_VEL
LIN {X 0,Y 376.007,Z 159.122,A -85,B 0,C 180,E1 -12401.473,E2 -12401.473} C_VEL
LIN {X 0,Y 376.056,Z 159.14,A -85,B 0,C 180,E1 -12404.832,E2 -12404.832} C_VEL
LIN {X 0,Y 376.047,Z 159.134,A -85,B 0,C 180,E1 -12408.136,E2 -12408.136} C_VEL
LIN {X 0,Y 376.218,Z 159.103,A -85,B 0,C 180,E1 -12411.917,E2 -12411.917} C_VEL
LIN {X 0,Y 376.168,Z 159.13,A -85,B 0,C 180,E1 -12414.639,E2 -12414.639} C_VEL
LIN {X 0,Y 376.348,Z 159.098,A -85,B 0,C 180,E1 -12417.859,E2 -12417.859} C_VEL
LIN {X 0,Y 376.483,Z 159.061,A -85,B 0,C 180,E1 -12419.999,E2 -12419.999} C_VEL
LIN {X 0,Y 376.186,Z 159.119,A -85,B 0,C 180,E1 -12423.212,E2 -12423.212} C_VEL
LIN {X 0,Y 376.231,Z 159.114,A -85,B 0,C 180,E1 -12426.609,E2 -12426.609} C_VEL
LIN {X 0,Y 376.202,Z 159.102,A -85,B 0,C 180,E1 -12428.595,E2 -12428.595} C_VEL
LIN {X 0,Y 376.045,Z 159.129,A -85,B 0,C 180,E1 -12431.863,E2 -12431.863} C_VEL
LIN {X 0,Y 376.054,Z 159.14,A -85,B 0,C 180,E1 -12435.167,E2 -12435.167} C_VEL
LIN {X 0,Y 376.004,Z 159.122,A -85,B 0,C 180,E1 -12438.526,E2 -12438.526} C_VEL
LIN {X 0,Y 375.959,Z 159.152,A -85,B 0,C 180,E1 -12441.954,E2 -12441.954} C_VEL
LIN {X 0,Y 376.002,Z 159.141,A -85,B 0,C 180,E1 -12445.461,E2 -12445.461} C_VEL
LIN {X 0,Y 375.971,Z 159.143,A -85,B 0,C 180,E1 -12449.078,E2 -12449.078} C_VEL
LIN {X 0,Y 375.945,Z 159.152,A -85,B 0,C 180,E1 -12452.828,E2 -12452.828} C_VEL
LIN {X 0,Y 375.953,Z 159.141,A -85,B 0,C 180,E1 -12455.415,E2 -12455.415} C_VEL
LIN {X 0,Y 375.971,Z 159.151,A -85,B 0,C 180,E1 -12458.271,E2 -12458.271} C_VEL
LIN {X 0,Y 375.93,Z 159.151,A -85,B 0,C 180,E1 -12461.601,E2 -12461.601} C_VEL
LIN {X 0,Y 375.95,Z 159.143,A -85,B 0,C 180,E1 -12465.264,E2 -12465.264} C_VEL
LIN {X 0,Y 375.935,Z 159.125,A -85,B 0,C 180,E1 -12469.133,E2 -12469.133} C_VEL
LIN {X 0,Y 375.961,Z 159.153,A -85,B 0,C 180,E1 -12471.912,E2 -12471.912} C_VEL
LIN {X 0,Y 375.975,Z 159.127,A -85,B 0,C 180,E1 -12475.333,E2 -12475.333} C_VEL
LIN {X 0,Y 375.973,Z 159.154,A -85,B 0,C 180,E1 -12478.44,E2 -12478.44} C_VEL
LIN {X 0,Y 375.998,Z 159.146,A -85,B 0,C 180,E1 -12482.142,E2 -12482.142} C_VEL
LIN {X 0,Y 376.002,Z 159.151,A -85,B 0,C 180,E1 -12484.539,E2 -12484.539} C_VEL
LIN {X 0,Y 375.959,Z 159.156,A -85,B 0,C 180,E1 -12488.046,E2 -12488.046} C_VEL
LIN {X 0,Y 376.02,Z 159.149,A -85,B 0,C 180,E1 -12491.474,E2 -12491.474} C_VEL
LIN {X 0,Y 376.054,Z 159.144,A -85,B 0,C 180,E1 -12494.833,E2 -12494.833} C_VEL
LIN {X 0,Y 376.115,Z 159.431,A -85,B 0,C 180,E1 -12496.109,E2 -12496.109} C_VEL
LIN {X 0,Y 376.404,Z 160.523,A -85,B 0,C 180,E1 -12496.467,E2 -12496.467} C_VEL
LIN {X 0,Y 377.861,Z 163.024,A -85,B 0,C 180,E1 -12497.103,E2 -12497.103} C_VEL
LIN {X 0,Y 380.043,Z 164.683,A -85,B 0,C 180,E1 -12497.945,E2 -12497.945} C_VEL
LIN {X 0,Y 381.205,Z 165.432,A -85,B 0,C 180,E1 -12498.434,E2 -12498.434} C_VEL
LIN {X 0,Y 382.765,Z 167.993,A -85,B 0,C 180,E1 -12499.152,E2 -12499.152} C_VEL
LIN {X 0,Y 385.027,Z 170.222,A -85,B 0,C 180,E1 -12500.287,E2 -12500.287} C_VEL
LIN {X 0,Y 387.591,Z 171.68,A -85,B 0,C 180,E1 -12501.659,E2 -12501.659} C_VEL
LIN {X 0,Y 389.285,Z 174.435,A -85,B 0,C 180,E1 -12502.841,E2 -12502.841} C_VEL
LIN {X 0,Y 391.041,Z 176.14,A -85,B 0,C 180,E1 -12504.198,E2 -12504.198} C_VEL
LIN {X 0,Y 392.756,Z 177.219,A -85,B 0,C 180,E1 -12505.896,E2 -12505.896} C_VEL
LIN {X 0,Y 393.915,Z 177.6,A -85,B 0,C 180,E1 -12507.579,E2 -12507.579} C_VEL
LIN {X 0,Y 394.407,Z 178.003,A -85,B 0,C 180,E1 -12508.979,E2 -12508.979} C_VEL
LIN {X 0,Y 394.593,Z 177.943,A -85,B 0,C 180,E1 -12510,E2 -12510} C_VEL
LIN {X 0,Y 394.096,Z 177.716,A -85,B 0,C 180,E1 -12512.044,E2 -12512.044} C_VEL
LIN {X 0,Y 393.066,Z 177.319,A -85,B 0,C 180,E1 -12513.725,E2 -12513.725} C_VEL
LIN {X 0,Y 391.609,Z 176.583,A -85,B 0,C 180,E1 -12515.277,E2 -12515.277} C_VEL
LIN {X 0,Y 389.867,Z 175.113,A -85,B 0,C 180,E1 -12516.729,E2 -12516.729} C_VEL
LIN {X 0,Y 388.033,Z 172.482,A -85,B 0,C 180,E1 -12518.061,E2 -12518.061} C_VEL
LIN {X 0,Y 387.368,Z 171.385,A -85,B 0,C 180,E1 -12518.477,E2 -12518.477} C_VEL
LIN {X 0,Y 384.676,Z 169.97,A -85,B 0,C 180,E1 -12519.88,E2 -12519.88} C_VEL
LIN {X 0,Y 382.443,Z 167.627,A -85,B 0,C 180,E1 -12520.991,E2 -12520.991} C_VEL
LIN {X 0,Y 380.868,Z 165.114,A -85,B 0,C 180,E1 -12521.711,E2 -12521.711} C_VEL
LIN {X 0,Y 378.262,Z 163.429,A -85,B 0,C 180,E1 -12522.746,E2 -12522.746} C_VEL
LIN {X 0,Y 376.574,Z 160.986,A -85,B 0,C 180,E1 -12523.445,E2 -12523.445} C_VEL
LIN {X 0,Y 376.2,Z 159.746,A -85,B 0,C 180,E1 -12523.73,E2 -12523.73} C_VEL
LIN {X 0,Y 376.064,Z 159.166,A -85,B 0,C 180,E1 -12524.337,E2 -12524.337} C_VEL
LIN {X 0,Y 376.04,Z 159.146,A -85,B 0,C 180,E1 -12527.607,E2 -12527.607} C_VEL
LIN {X 0,Y 375.974,Z 159.154,A -85,B 0,C 180,E1 -12530.832,E2 -12530.832} C_VEL
LIN {X 0,Y 375.99,Z 159.15,A -85,B 0,C 180,E1 -12534.281,E2 -12534.281} C_VEL
LIN {X 0,Y 376.015,Z 159.148,A -85,B 0,C 180,E1 -12536.652,E2 -12536.652} C_VEL
LIN {X 0,Y 375.972,Z 159.136,A -85,B 0,C 180,E1 -12539.079,E2 -12539.079} C_VEL
LIN {X 0,Y 375.957,Z 159.147,A -85,B 0,C 180,E1 -12542.827,E2 -12542.827} C_VEL
LIN {X 0,Y 375.953,Z 159.134,A -85,B 0,C 180,E1 -12545.415,E2 -12545.415} C_VEL
LIN {X 0,Y 375.971,Z 159.153,A -85,B 0,C 180,E1 -12548.271,E2 -12548.271} C_VEL
LIN {X 0,Y 375.978,Z 159.137,A -85,B 0,C 180,E1 -12550.022,E2 -12550.022} C_VEL
LIN {X 0,Y 375.244,Z 159.21,A -85,B 0,C 180,E1 -12550.916,E2 -12550.916} C_VEL
LIN {X 0,Y 372.337,Z 159.564,A -85,B 0,C 180,E1 -12552.368,E2 -12552.368} C_VEL
LIN {X 0,Y 369.94,Z 159.876,A -85,B 0,C 180,E1 -12553.542,E2 -12553.542} C_VEL
LIN {X 0,Y 368.956,Z 160.011,A -85,B 0,C 180,E1 -12554.451,E2 -12554.451} C_VEL
LIN {X 0,Y 368.898,Z 160.021,A -85,B 0,C 180,E1 -12554.758,E2 -12554.758} C_VEL
LIN {X 0,Y 368.878,Z 160.032,A -85,B 0,C 180,E1 -12558.178,E2 -12558.178} C_VEL
LIN {X 0,Y 368.905,Z 160.032,A -85,B 0,C 180,E1 -12561.36,E2 -12561.36} C_VEL
LIN {X 0,Y 368.932,Z 160.01,A -85,B 0,C 180,E1 -12565.147,E2 -12565.147} C_VEL
LIN {X 0,Y 368.924,Z 160.029,A -85,B 0,C 180,E1 -12569.047,E2 -12569.047} C_VEL
LIN {X 0,Y 368.982,Z 160.012,A -85,B 0,C 180,E1 -12571.565,E2 -12571.565} C_VEL
LIN {X 0,Y 368.953,Z 160.022,A -85,B 0,C 180,E1 -12575.225,E2 -12575.225} C_VEL
LIN {X 0,Y 368.933,Z 160.018,A -85,B 0,C 180,E1 -12578.974,E2 -12578.974} C_VEL
LIN {X 0,Y 368.986,Z 160.004,A -85,B 0,C 180,E1 -12582.258,E2 -12582.258} C_VEL
LIN {X 0,Y 369.033,Z 160.015,A -85,B 0,C 180,E1 -12586.228,E2 -12586.228} C_VEL
LIN {X 0,Y 369.063,Z 159.985,A -85,B 0,C 180,E1 -12590.132,E2 -12590.132} C_VEL
LIN {X 0,Y 369.185,Z 159.989,A -85,B 0,C 180,E1 -12592.343,E2 -12592.343} C_VEL
LIN {X 0,Y 369.141,Z 160.001,A -85,B 0,C 180,E1 -12594.538,E2 -12594.538} C_VEL
LIN {X 0,Y 369.315,Z 159.966,A -85,B 0,C 180,E1 -12597.819,E2 -12597.819} C_VEL
LIN {X 0,Y 369.453,Z 159.936,A -85,B 0,C 180,E1 -12600.001,E2 -12600.001} C_VEL
LIN {X 0,Y 369.313,Z 159.974,A -85,B 0,C 180,E1 -12602.182,E2 -12602.182} C_VEL
LIN {X 0,Y 369.2,Z 159.99,A -85,B 0,C 180,E1 -12606.559,E2 -12606.559} C_VEL
LIN {X 0,Y 369.065,Z 159.984,A -85,B 0,C 180,E1 -12609.869,E2 -12609.869} C_VEL
LIN {X 0,Y 369.035,Z 160.014,A -85,B 0,C 180,E1 -12613.773,E2 -12613.773} C_VEL
LIN {X 0,Y 368.999,Z 159.997,A -85,B 0,C 180,E1 -12617.769,E2 -12617.769} C_VEL
LIN {X 0,Y 368.928,Z 160.022,A -85,B 0,C 180,E1 -12621.22,E2 -12621.22} C_VEL
LIN {X 0,Y 368.956,Z 160.02,A -85,B 0,C 180,E1 -12624.776,E2 -12624.776} C_VEL
LIN {X 0,Y 368.962,Z 160.005,A -85,B 0,C 180,E1 -12627.204,E2 -12627.204} C_VEL
LIN {X 0,Y 368.928,Z 160.031,A -85,B 0,C 180,E1 -12630.954,E2 -12630.954} C_VEL
LIN {X 0,Y 368.928,Z 160.017,A -85,B 0,C 180,E1 -12635.002,E2 -12635.002} C_VEL
LIN {X 0,Y 368.906,Z 160.028,A -85,B 0,C 180,E1 -12638.641,E2 -12638.641} C_VEL
LIN {X 0,Y 368.881,Z 160.033,A -85,B 0,C 180,E1 -12642.01,E2 -12642.01} C_VEL
LIN {X 0,Y 368.88,Z 160.032,A -85,B 0,C 180,E1 -12645.176,E2 -12645.176} C_VEL
LIN {X 0,Y 368.883,Z 160.025,A -85,B 0,C 180,E1 -12648.178,E2 -12648.178} C_VEL
LIN {X 0,Y 368.911,Z 160.027,A -85,B 0,C 180,E1 -12651.36,E2 -12651.36} C_VEL
LIN {X 0,Y 368.938,Z 160.018,A -85,B 0,C 180,E1 -12655.147,E2 -12655.147} C_VEL
LIN {X 0,Y 368.972,Z 160.191,A -85,B 0,C 180,E1 -12658.777,E2 -12658.777} C_VEL
LIN {X 0,Y 370.708,Z 168.867,A -85,B 0,C 180,E1 -12661.709,E2 -12661.709} C_VEL
LIN {X 0,Y 371.905,Z 176.18,A -85,B 0,C 180,E1 -12663.937,E2 -12663.937} C_VEL
LIN {X 0,Y 371.315,Z 183.294,A -85,B 0,C 180,E1 -12665.988,E2 -12665.988} C_VEL
LIN {X 0,Y 370.584,Z 191.151,A -85,B 0,C 180,E1 -12668.271,E2 -12668.271} C_VEL
LIN {X 0,Y 371.483,Z 195.852,A -85,B 0,C 180,E1 -12668.476,E2 -12668.476} C_VEL
LIN {X 0,Y 376.707,Z 223.99,A -85,B 0,C 180,E1 -12669.348,E2 -12669.348} C_VEL
LIN {X 0,Y 375.685,Z 295.981,A -85,B 0,C 180,E1 -12670.749,E2 -12670.749} C_VEL
LIN {X 0,Y 375.252,Z 306.75,A -85,B 0,C 180,E1 -12671.081,E2 -12671.081} C_VEL
LIN {X 0,Y 374.714,Z 315.85,A -85,B 0,C 180,E1 -12671.478,E2 -12671.478} C_VEL
LIN {X 0,Y 374.067,Z 325.204,A -85,B 0,C 180,E1 -12672.012,E2 -12672.012} C_VEL
LIN {X 0,Y 373.189,Z 335.343,A -85,B 0,C 180,E1 -12672.746,E2 -12672.746} C_VEL
LIN {X 0,Y 372.368,Z 344.339,A -85,B 0,C 180,E1 -12673.554,E2 -12673.554} C_VEL
LIN {X 0,Y 371.474,Z 353.067,A -85,B 0,C 180,E1 -12674.5,E2 -12674.5} C_VEL
LIN {X 0,Y 370.744,Z 360.789,A -85,B 0,C 180,E1 -12675.501,E2 -12675.501} C_VEL
LIN {X 0,Y 370.083,Z 367.684,A -85,B 0,C 180,E1 -12676.548,E2 -12676.548} C_VEL
LIN {X 0,Y 369.423,Z 373.886,A -85,B 0,C 180,E1 -12677.642,E2 -12677.642} C_VEL
LIN {X 0,Y 368.673,Z 380.421,A -85,B 0,C 180,E1 -12679.011,E2 -12679.011} C_VEL
LIN {X 0,Y 368.285,Z 384.924,A -85,B 0,C 180,E1 -12680.111,E2 -12680.111} C_VEL
LIN {X 0,Y 367.841,Z 390.415,A -85,B 0,C 180,E1 -12681.761,E2 -12681.761} C_VEL
LIN {X 0,Y 367.565,Z 394.74,A -85,B 0,C 180,E1 -12683.412,E2 -12683.412} C_VEL
LIN {X 0,Y 367.465,Z 397.107,A -85,B 0,C 180,E1 -12684.513,E2 -12684.513} C_VEL
LIN {X 0,Y 367.437,Z 398.907,A -85,B 0,C 180,E1 -12685.612,E2 -12685.612} C_VEL
LIN {X 0,Y 367.36,Z 401.35,A -85,B 0,C 180,E1 -12687.807,E2 -12687.807} C_VEL
LIN {X 0,Y 367.404,Z 401.94,A -85,B 0,C 180,E1 -12688.904,E2 -12688.904} C_VEL
LIN {X 0,Y 367.404,Z 401.94,A -85,B 0,C 180,E1 -12691.096,E2 -12691.096} C_VEL
LIN {X 0,Y 367.36,Z 401.35,A -85,B 0,C 180,E1 -12692.193,E2 -12692.193} C_VEL
LIN {X 0,Y 367.437,Z 398.907,A -85,B 0,C 180,E1 -12694.388,E2 -12694.388} C_VEL
LIN {X 0,Y 367.48,Z 396.015,A -85,B 0,C 180,E1 -12696.012,E2 -12696.012} C_VEL
LIN {X 0,Y 367.718,Z 391.969,A -85,B 0,C 180,E1 -12697.688,E2 -12697.688} C_VEL
LIN {X 0,Y 368.11,Z 386.839,A -85,B 0,C 180,E1 -12699.339,E2 -12699.339} C_VEL
LIN {X 0,Y 368.587,Z 381.577,A -85,B 0,C 180,E1 -12700.714,E2 -12700.714} C_VEL
LIN {X 0,Y 369.247,Z 375.261,A -85,B 0,C 180,E1 -12702.085,E2 -12702.085} C_VEL
LIN {X 0,Y 369.91,Z 369.311,A -85,B 0,C 180,E1 -12703.179,E2 -12703.179} C_VEL
LIN {X 0,Y 370.561,Z 362.382,A -85,B 0,C 180,E1 -12704.274,E2 -12704.274} C_VEL
LIN {X 0,Y 371.392,Z 354.202,A -85,B 0,C 180,E1 -12705.362,E2 -12705.362} C_VEL
LIN {X 0,Y 372.207,Z 345.69,A -85,B 0,C 180,E1 -12706.312,E2 -12706.312} C_VEL
LIN {X 0,Y 373.047,Z 336.975,A -85,B 0,C 180,E1 -12707.119,E2 -12707.119} C_VEL
LIN {X 0,Y 373.843,Z 327.217,A -85,B 0,C 180,E1 -12707.858,E2 -12707.858} C_VEL
LIN {X 0,Y 374.531,Z 318.424,A -85,B 0,C 180,E1 -12708.39,E2 -12708.39} C_VEL
LIN {X 0,Y 375.126,Z 308.497,A -85,B 0,C 180,E1 -12708.855,E2 -12708.855} C_VEL
LIN {X 0,Y 375.615,Z 298.645,A -85,B 0,C 180,E1 -12709.184,E2 -12709.184} C_VEL
LIN {X 0,Y 376.141,Z 273.179,A -85,B 0,C 180,E1 -12709.705,E2 -12709.705} C_VEL
LIN {X 0,Y 376.623,Z 223.785,A -85,B 0,C 180,E1 -12710.661,E2 -12710.661} C_VEL
LIN {X 0,Y 371.576,Z 196.268,A -85,B 0,C 180,E1 -12711.51,E2 -12711.51} C_VEL
LIN {X 0,Y 370.557,Z 191.243,A -85,B 0,C 180,E1 -12711.716,E2 -12711.716} C_VEL
LIN {X 0,Y 370.875,Z 187.195,A -85,B 0,C 180,E1 -12712.859,E2 -12712.859} C_VEL
LIN {X 0,Y 372.006,Z 177.348,A -85,B 0,C 180,E1 -12715.754,E2 -12715.754} C_VEL
LIN {X 0,Y 371.467,Z 172.597,A -85,B 0,C 180,E1 -12717.224,E2 -12717.224} C_VEL
LIN {X 0,Y 369.321,Z 161.975,A -85,B 0,C 180,E1 -12720.599,E2 -12720.599} C_VEL
LIN {X 0,Y 368.928,Z 160.044,A -85,B 0,C 180,E1 -12721.351,E2 -12721.351} C_VEL
LIN {X 0,Y 368.93,Z 160.018,A -85,B 0,C 180,E1 -12725.001,E2 -12725.001} C_VEL
LIN {X 0,Y 368.911,Z 160.027,A -85,B 0,C 180,E1 -12728.64,E2 -12728.64} C_VEL
LIN {X 0,Y 368.882,Z 160.028,A -85,B 0,C 180,E1 -12732.009,E2 -12732.009} C_VEL
LIN {X 0,Y 368.88,Z 160.03,A -85,B 0,C 180,E1 -12735.175,E2 -12735.175} C_VEL
LIN {X 0,Y 368.882,Z 160.033,A -85,B 0,C 180,E1 -12738.177,E2 -12738.177} C_VEL
LIN {X 0,Y 368.906,Z 160.028,A -85,B 0,C 180,E1 -12741.359,E2 -12741.359} C_VEL
LIN {X 0,Y 368.936,Z 160.015,A -85,B 0,C 180,E1 -12745.146,E2 -12745.146} C_VEL
LIN {X 0,Y 368.928,Z 160.031,A -85,B 0,C 180,E1 -12749.046,E2 -12749.046} C_VEL
LIN {X 0,Y 368.962,Z 160.005,A -85,B 0,C 180,E1 -12752.796,E2 -12752.796} C_VEL
LIN {X 0,Y 368.944,Z 160.023,A -85,B 0,C 180,E1 -12756.112,E2 -12756.112} C_VEL
LIN {X 0,Y 368.935,Z 160.012,A -85,B 0,C 180,E1 -12759.946,E2 -12759.946} C_VEL
LIN {X 0,Y 368.974,Z 160.016,A -85,B 0,C 180,E1 -12763.398,E2 -12763.398} C_VEL
LIN {X 0,Y 369.055,Z 160.01,A -85,B 0,C 180,E1 -12766.79,E2 -12766.79} C_VEL
LIN {X 0,Y 369.065,Z 159.984,A -85,B 0,C 180,E1 -12770.131,E2 -12770.131} C_VEL
LIN {X 0,Y 369.2,Z 159.99,A -85,B 0,C 180,E1 -12773.441,E2 -12773.441} C_VEL
LIN {X 0,Y 369.313,Z 159.974,A -85,B 0,C 180,E1 -12777.818,E2 -12777.818} C_VEL
LIN {X 0,Y 369.453,Z 159.936,A -85,B 0,C 180,E1 -12779.999,E2 -12779.999} C_VEL
LIN {X 0,Y 369.315,Z 159.966,A -85,B 0,C 180,E1 -12782.181,E2 -12782.181} C_VEL
LIN {X 0,Y 369.202,Z 159.99,A -85,B 0,C 180,E1 -12786.597,E2 -12786.597} C_VEL
LIN {X 0,Y 369.134,Z 159.981,A -85,B 0,C 180,E1 -12788.76,E2 -12788.76} C_VEL
LIN {X 0,Y 369.001,Z 160.009,A -85,B 0,C 180,E1 -12792.093,E2 -12792.093} C_VEL
LIN {X 0,Y 368.993,Z 160.021,A -85,B 0,C 180,E1 -12795.464,E2 -12795.464} C_VEL
LIN {X 0,Y 368.954,Z 159.999,A -85,B 0,C 180,E1 -12798.894,E2 -12798.894} C_VEL
LIN {X 0,Y 368.928,Z 160.028,A -85,B 0,C 180,E1 -12802.395,E2 -12802.395} C_VEL
LIN {X 0,Y 368.995,Z 160.006,A -85,B 0,C 180,E1 -12805.98,E2 -12805.98} C_VEL
LIN {X 0,Y 368.962,Z 160.015,A -85,B 0,C 180,E1 -12808.813,E2 -12808.813} C_VEL
LIN {X 0,Y 368.894,Z 160.03,A -85,B 0,C 180,E1 -12812.238,E2 -12812.238} C_VEL
LIN {X 0,Y 368.924,Z 160.012,A -85,B 0,C 180,E1 -12815.001,E2 -12815.001} C_VEL
LIN {X 0,Y 368.905,Z 160.032,A -85,B 0,C 180,E1 -12818.64,E2 -12818.64} C_VEL
LIN {X 0,Y 368.877,Z 160.033,A -85,B 0,C 180,E1 -12822.009,E2 -12822.009} C_VEL
LIN {X 0,Y 368.903,Z 160.022,A -85,B 0,C 180,E1 -12825.18,E2 -12825.18} C_VEL
LIN {X 0,Y 368.877,Z 159.993,A -85,B 0,C 180,E1 -12828.177,E2 -12828.177} C_VEL
LIN {X 0,Y 368.905,Z 160.034,A -85,B 0,C 180,E1 -12831.359,E2 -12831.359} C_VEL
LIN {X 0,Y 368.932,Z 160.003,A -85,B 0,C 180,E1 -12835.146,E2 -12835.146} C_VEL
LIN {X 0,Y 368.925,Z 160.026,A -85,B 0,C 180,E1 -12839.046,E2 -12839.046} C_VEL
LIN {X 0,Y 368.982,Z 160.011,A -85,B 0,C 180,E1 -12841.565,E2 -12841.565} C_VEL
LIN {X 0,Y 368.953,Z 160.028,A -85,B 0,C 180,E1 -12845.225,E2 -12845.225} C_VEL
LIN {X 0,Y 368.933,Z 160.031,A -85,B 0,C 180,E1 -12848.973,E2 -12848.973} C_VEL
LIN {X 0,Y 368.986,Z 160.025,A -85,B 0,C 180,E1 -12852.257,E2 -12852.257} C_VEL
LIN {X 0,Y 369.013,Z 160.292,A -85,B 0,C 180,E1 -12854.04,E2 -12854.04} C_VEL
LIN {X 0,Y 369.277,Z 161.285,A -85,B 0,C 180,E1 -12854.353,E2 -12854.353} C_VEL
LIN {X 0,Y 370.509,Z 163.579,A -85,B 0,C 180,E1 -12854.811,E2 -12854.811} C_VEL
LIN {X 0,Y 372.883,Z 165.491,A -85,B 0,C 180,E1 -12855.608,E2 -12855.608} C_VEL
LIN {X 0,Y 373.911,Z 166.227,A -85,B 0,C 180,E1 -12855.94,E2 -12855.94} C_VEL
LIN {X 0,Y 375.803,Z 169.293,A -85,B 0,C 180,E1 -12856.694,E2 -12856.694} C_VEL
LIN {X 0,Y 378.433,Z 171.423,A -85,B 0,C 180,E1 -12857.668,E2 -12857.668} C_VEL
LIN {X 0,Y 379.535,Z 172.197,A -85,B 0,C 180,E1 -12858.132,E2 -12858.132} C_VEL
LIN {X 0,Y 381.399,Z 174.937,A -85,B 0,C 180,E1 -12858.979,E2 -12858.979} C_VEL
LIN {X 0,Y 383.941,Z 177.232,A -85,B 0,C 180,E1 -12860.208,E2 -12860.208} C_VEL
LIN {X 0,Y 386.289,Z 178.546,A -85,B 0,C 180,E1 -12861.433,E2 -12861.433} C_VEL
LIN {X 0,Y 388.224,Z 181.442,A -85,B 0,C 180,E1 -12862.72,E2 -12862.72} C_VEL
LIN {X 0,Y 390.286,Z 183.324,A -85,B 0,C 180,E1 -12864.316,E2 -12864.316} C_VEL
LIN {X 0,Y 391.883,Z 184.245,A -85,B 0,C 180,E1 -12865.886,E2 -12865.886} C_VEL
LIN {X 0,Y 392.994,Z 184.615,A -85,B 0,C 180,E1 -12867.456,E2 -12867.456} C_VEL
LIN {X 0,Y 393.545,Z 185.049,A -85,B 0,C 180,E1 -12868.977,E2 -12868.977} C_VEL
LIN {X 0,Y 393.727,Z 184.99,A -85,B 0,C 180,E1 -12870,E2 -12870} C_VEL
LIN {X 0,Y 393.467,Z 184.922,A -85,B 0,C 180,E1 -12871.535,E2 -12871.535} C_VEL
LIN {X 0,Y 392.738,Z 184.495,A -85,B 0,C 180,E1 -12873.077,E2 -12873.077} C_VEL
LIN {X 0,Y 391.175,Z 183.885,A -85,B 0,C 180,E1 -12874.896,E2 -12874.896} C_VEL
LIN {X 0,Y 389.129,Z 182.375,A -85,B 0,C 180,E1 -12876.62,E2 -12876.62} C_VEL
LIN {X 0,Y 387.407,Z 180.295,A -85,B 0,C 180,E1 -12877.871,E2 -12877.871} C_VEL
LIN {X 0,Y 385.95,Z 178.186,A -85,B 0,C 180,E1 -12878.772,E2 -12878.772} C_VEL
LIN {X 0,Y 383.231,Z 176.734,A -85,B 0,C 180,E1 -12880.134,E2 -12880.134} C_VEL
LIN {X 0,Y 380.895,Z 174.359,A -85,B 0,C 180,E1 -12881.238,E2 -12881.238} C_VEL
LIN {X 0,Y 379.161,Z 171.786,A -85,B 0,C 180,E1 -12882.036,E2 -12882.036} C_VEL
LIN {X 0,Y 376.571,Z 170.1,A -85,B 0,C 180,E1 -12883.011,E2 -12883.011} C_VEL
LIN {X 0,Y 374.518,Z 167.352,A -85,B 0,C 180,E1 -12883.833,E2 -12883.833} C_VEL
LIN {X 0,Y 373.644,Z 165.876,A -85,B 0,C 180,E1 -12884.153,E2 -12884.153} C_VEL
LIN {X 0,Y 370.852,Z 163.969,A -85,B 0,C 180,E1 -12885.068,E2 -12885.068} C_VEL
LIN {X 0,Y 369.45,Z 161.788,A -85,B 0,C 180,E1 -12885.569,E2 -12885.569} C_VEL
LIN {X 0,Y 369.037,Z 160.424,A -85,B 0,C 180,E1 -12885.888,E2 -12885.888} C_VEL
LIN {X 0,Y 368.972,Z 160.026,A -85,B 0,C 180,E1 -12886.601,E2 -12886.601} C_VEL
LIN {X 0,Y 368.933,Z 160.031,A -85,B 0,C 180,E1 -12890.053,E2 -12890.053} C_VEL
LIN {X 0,Y 368.941,Z 160.03,A -85,B 0,C 180,E1 -12893.887,E2 -12893.887} C_VEL
LIN {X 0,Y 368.967,Z 160.028,A -85,B 0,C 180,E1 -12897.203,E2 -12897.203} C_VEL
LIN {X 0,Y 368.92,Z 160.014,A -85,B 0,C 180,E1 -12899.69,E2 -12899.69} C_VEL
LIN {X 0,Y 368.897,Z 160.016,A -85,B 0,C 180,E1 -12903.538,E2 -12903.538} C_VEL
LIN {X 0,Y 368.898,Z 160.028,A -85,B 0,C 180,E1 -12906.856,E2 -12906.856} C_VEL
LIN {X 0,Y 368.905,Z 160.008,A -85,B 0,C 180,E1 -12910.37,E2 -12910.37} C_VEL
LIN {X 0,Y 368.879,Z 160.009,A -85,B 0,C 180,E1 -12913.616,E2 -12913.616} C_VEL
LIN {X 0,Y 368.898,Z 160.021,A -85,B 0,C 180,E1 -12914.758,E2 -12914.758} C_VEL
LIN {X 0,Y 368.281,Z 160.111,A -85,B 0,C 180,E1 -12915.669,E2 -12915.669} C_VEL
LIN {X 0,Y 365.414,Z 160.467,A -85,B 0,C 180,E1 -12917.15,E2 -12917.15} C_VEL
LIN {X 0,Y 362.957,Z 160.766,A -85,B 0,C 180,E1 -12918.348,E2 -12918.348} C_VEL
LIN {X 0,Y 361.908,Z 160.89,A -85,B 0,C 180,E1 -12919.275,E2 -12919.275} C_VEL
LIN {X 0,Y 361.828,Z 160.9,A -85,B 0,C 180,E1 -12919.589,E2 -12919.589} C_VEL
LIN {X 0,Y 361.868,Z 160.908,A -85,B 0,C 180,E1 -12922.983,E2 -12922.983} C_VEL
LIN {X 0,Y 361.854,Z 160.899,A -85,B 0,C 180,E1 -12926.631,E2 -12926.631} C_VEL
LIN {X 0,Y 361.871,Z 160.908,A -85,B 0,C 180,E1 -12929.673,E2 -12929.673} C_VEL
LIN {X 0,Y 361.95,Z 160.88,A -85,B 0,C 180,E1 -12933.476,E2 -12933.476} C_VEL
LIN {X 0,Y 361.886,Z 160.904,A -85,B 0,C 180,E1 -12937.145,E2 -12937.145} C_VEL
LIN {X 0,Y 361.902,Z 160.877,A -85,B 0,C 180,E1 -12940.724,E2 -12940.724} C_VEL
LIN {X 0,Y 361.928,Z 160.892,A -85,B 0,C 180,E1 -12943.066,E2 -12943.066} C_VEL
LIN {X 0,Y 361.995,Z 160.889,A -85,B 0,C 180,E1 -12946.528,E2 -12946.528} C_VEL
LIN {X 0,Y 362.027,Z 160.861,A -85,B 0,C 180,E1 -12949.939,E2 -12949.939} C_VEL
LIN {X 0,Y 362.143,Z 160.862,A -85,B 0,C 180,E1 -12952.193,E2 -12952.193} C_VEL
LIN {X 0,Y 362.115,Z 160.877,A -85,B 0,C 180,E1 -12954.432,E2 -12954.432} C_VEL
LIN {X 0,Y 362.279,Z 160.842,A -85,B 0,C 180,E1 -12957.777,E2 -12957.777} C_VEL
LIN {X 0,Y 362.423,Z 160.81,A -85,B 0,C 180,E1 -12960.001,E2 -12960.001} C_VEL
LIN {X 0,Y 362.278,Z 160.85,A -85,B 0,C 180,E1 -12962.224,E2 -12962.224} C_VEL
LIN {X 0,Y 362.162,Z 160.867,A -85,B 0,C 180,E1 -12966.687,E2 -12966.687} C_VEL
LIN {X 0,Y 362.028,Z 160.861,A -85,B 0,C 180,E1 -12970.063,E2 -12970.063} C_VEL
LIN {X 0,Y 361.996,Z 160.89,A -85,B 0,C 180,E1 -12973.899,E2 -12973.899} C_VEL
LIN {X 0,Y 361.966,Z 160.872,A -85,B 0,C 180,E1 -12977.939,E2 -12977.939} C_VEL
LIN {X 0,Y 361.892,Z 160.902,A -85,B 0,C 180,E1 -12981.654,E2 -12981.654} C_VEL
LIN {X 0,Y 361.927,Z 160.888,A -85,B 0,C 180,E1 -12985.291,E2 -12985.291} C_VEL
LIN {X 0,Y 361.907,Z 160.888,A -85,B 0,C 180,E1 -12987.78,E2 -12987.78} C_VEL
LIN {X 0,Y 361.836,Z 160.91,A -85,B 0,C 180,E1 -12991.63,E2 -12991.63} C_VEL
LIN {X 0,Y 361.873,Z 160.9,A -85,B 0,C 180,E1 -12995.345,E2 -12995.345} C_VEL
LIN {X 0,Y 361.867,Z 160.901,A -85,B 0,C 180,E1 -12999.027,E2 -12999.027} C_VEL
LIN {X 0,Y 361.836,Z 160.913,A -85,B 0,C 180,E1 -13002.83,E2 -13002.83} C_VEL
LIN {X 0,Y 361.819,Z 160.914,A -85,B 0,C 180,E1 -13005.947,E2 -13005.947} C_VEL
LIN {X 0,Y 361.836,Z 160.891,A -85,B 0,C 180,E1 -13009.245,E2 -13009.245} C_VEL
LIN {X 0,Y 361.872,Z 160.908,A -85,B 0,C 180,E1 -13012.776,E2 -13012.776} C_VEL
LIN {X 0,Y 361.856,Z 160.907,A -85,B 0,C 180,E1 -13015.72,E2 -13015.72} C_VEL
LIN {X 0,Y 361.929,Z 161.106,A -85,B 0,C 180,E1 -13018.45,E2 -13018.45} C_VEL
LIN {X 0,Y 363.464,Z 168.684,A -85,B 0,C 180,E1 -13021.092,E2 -13021.092} C_VEL
LIN {X 0,Y 364.934,Z 177.047,A -85,B 0,C 180,E1 -13023.709,E2 -13023.709} C_VEL
LIN {X 0,Y 364.714,Z 181.149,A -85,B 0,C 180,E1 -13024.917,E2 -13024.917} C_VEL
LIN {X 0,Y 363.663,Z 191.014,A -85,B 0,C 180,E1 -13027.845,E2 -13027.845} C_VEL
LIN {X 0,Y 365.005,Z 197.568,A -85,B 0,C 180,E1 -13028.114,E2 -13028.114} C_VEL
LIN {X 0,Y 370.099,Z 225.16,A -85,B 0,C 180,E1 -13028.99,E2 -13028.99} C_VEL
LIN {X 0,Y 369.002,Z 295.793,A -85,B 0,C 180,E1 -13030.386,E2 -13030.386} C_VEL
LIN {X 0,Y 368.625,Z 305.685,A -85,B 0,C 180,E1 -13030.691,E2 -13030.691} C_VEL
LIN {X 0,Y 367.981,Z 315.658,A -85,B 0,C 180,E1 -13031.126,E2 -13031.126} C_VEL
LIN {X 0,Y 367.305,Z 325.012,A -85,B 0,C 180,E1 -13031.669,E2 -13031.669} C_VEL
LIN {X 0,Y 366.416,Z 335.152,A -85,B 0,C 180,E1 -13032.417,E2 -13032.417} C_VEL
LIN {X 0,Y 365.532,Z 344.147,A -85,B 0,C 180,E1 -13033.238,E2 -13033.238} C_VEL
LIN {X 0,Y 364.606,Z 352.874,A -85,B 0,C 180,E1 -13034.201,E2 -13034.201} C_VEL
LIN {X 0,Y 363.804,Z 361.011,A -85,B 0,C 180,E1 -13035.28,E2 -13035.28} C_VEL
LIN {X 0,Y 362.941,Z 369.118,A -85,B 0,C 180,E1 -13036.564,E2 -13036.564} C_VEL
LIN {X 0,Y 362.272,Z 375.068,A -85,B 0,C 180,E1 -13037.679,E2 -13037.679} C_VEL
LIN {X 0,Y 361.567,Z 381.384,A -85,B 0,C 180,E1 -13039.076,E2 -13039.076} C_VEL
LIN {X 0,Y 361.063,Z 386.647,A -85,B 0,C 180,E1 -13040.477,E2 -13040.477} C_VEL
LIN {X 0,Y 360.668,Z 391.777,A -85,B 0,C 180,E1 -13042.16,E2 -13042.16} C_VEL
LIN {X 0,Y 360.5,Z 394.548,A -85,B 0,C 180,E1 -13043.283,E2 -13043.283} C_VEL
LIN {X 0,Y 360.385,Z 396.915,A -85,B 0,C 180,E1 -13044.404,E2 -13044.404} C_VEL
LIN {X 0,Y 360.348,Z 398.715,A -85,B 0,C 180,E1 -13045.526,E2 -13045.526} C_VEL
LIN {X 0,Y 360.264,Z 401.159,A -85,B 0,C 180,E1 -13047.764,E2 -13047.764} C_VEL
LIN {X 0,Y 360.304,Z 401.748,A -85,B 0,C 180,E1 -13048.882,E2 -13048.882} C_VEL
LIN {X 0,Y 360.304,Z 401.748,A -85,B 0,C 180,E1 -13051.118,E2 -13051.118} C_VEL
LIN {X 0,Y 360.264,Z 401.159,A -85,B 0,C 180,E1 -13052.236,E2 -13052.236} C_VEL
LIN {X 0,Y 360.348,Z 398.715,A -85,B 0,C 180,E1 -13054.474,E2 -13054.474} C_VEL
LIN {X 0,Y 360.379,Z 396.189,A -85,B 0,C 180,E1 -13055.961,E2 -13055.961} C_VEL
LIN {X 0,Y 360.591,Z 393.308,A -85,B 0,C 180,E1 -13057.278,E2 -13057.278} C_VEL
LIN {X 0,Y 360.92,Z 388.563,A -85,B 0,C 180,E1 -13058.962,E2 -13058.962} C_VEL
LIN {X 0,Y 361.491,Z 382.541,A -85,B 0,C 180,E1 -13060.643,E2 -13060.643} C_VEL
LIN {X 0,Y 362.1,Z 376.444,A -85,B 0,C 180,E1 -13062.043,E2 -13062.043} C_VEL
LIN {X 0,Y 362.793,Z 370.745,A -85,B 0,C 180,E1 -13063.157,E2 -13063.157} C_VEL
LIN {X 0,Y 363.678,Z 362.19,A -85,B 0,C 180,E1 -13064.55,E2 -13064.55} C_VEL
LIN {X 0,Y 364.526,Z 354.01,A -85,B 0,C 180,E1 -13065.659,E2 -13065.659} C_VEL
LIN {X 0,Y 365.383,Z 345.498,A -85,B 0,C 180,E1 -13066.625,E2 -13066.625} C_VEL
LIN {X 0,Y 366.246,Z 336.783,A -85,B 0,C 180,E1 -13067.447,E2 -13067.447} C_VEL
LIN {X 0,Y 367.099,Z 327.025,A -85,B 0,C 180,E1 -13068.198,E2 -13068.198} C_VEL
LIN {X 0,Y 367.894,Z 316.945,A -85,B 0,C 180,E1 -13068.806,E2 -13068.806} C_VEL
LIN {X 0,Y 368.495,Z 307.432,A -85,B 0,C 180,E1 -13069.244,E2 -13069.244} C_VEL
LIN {X 0,Y 368.959,Z 297.122,A -85,B 0,C 180,E1 -13069.58,E2 -13069.58} C_VEL
LIN {X 0,Y 369.789,Z 249.786,A -85,B 0,C 180,E1 -13070.528,E2 -13070.528} C_VEL
LIN {X 0,Y 370.011,Z 224.71,A -85,B 0,C 180,E1 -13071.025,E2 -13071.025} C_VEL
LIN {X 0,Y 364.895,Z 197.088,A -85,B 0,C 180,E1 -13071.903,E2 -13071.903} C_VEL
LIN {X 0,Y 363.653,Z 191.179,A -85,B 0,C 180,E1 -13072.136,E2 -13072.136} C_VEL
LIN {X 0,Y 363.795,Z 188.918,A -85,B 0,C 180,E1 -13072.729,E2 -13072.729} C_VEL
LIN {X 0,Y 365.034,Z 178.166,A -85,B 0,C 180,E1 -13075.976,E2 -13075.976} C_VEL
LIN {X 0,Y 364.148,Z 172.116,A -85,B 0,C 180,E1 -13077.906,E2 -13077.906} C_VEL
LIN {X 0,Y 362.35,Z 163.274,A -85,B 0,C 180,E1 -13080.789,E2 -13080.789} C_VEL
LIN {X 0,Y 361.912,Z 160.967,A -85,B 0,C 180,E1 -13081.622,E2 -13081.622} C_VEL
LIN {X 0,Y 361.87,Z 160.895,A -85,B 0,C 180,E1 -13085.636,E2 -13085.636} C_VEL
LIN {X 0,Y 361.872,Z 160.896,A -85,B 0,C 180,E1 -13089.026,E2 -13089.026} C_VEL
LIN {X 0,Y 361.837,Z 160.911,A -85,B 0,C 180,E1 -13092.828,E2 -13092.828} C_VEL
LIN {X 0,Y 361.818,Z 160.912,A -85,B 0,C 180,E1 -13095.946,E2 -13095.946} C_VEL
LIN {X 0,Y 361.835,Z 160.906,A -85,B 0,C 180,E1 -13099.244,E2 -13099.244} C_VEL
LIN {X 0,Y 361.862,Z 160.909,A -85,B 0,C 180,E1 -13102.777,E2 -13102.777} C_VEL
LIN {X 0,Y 361.853,Z 160.893,A -85,B 0,C 180,E1 -13105.719,E2 -13105.719} C_VEL
LIN {X 0,Y 361.872,Z 160.907,A -85,B 0,C 180,E1 -13109.671,E2 -13109.671} C_VEL
LIN {X 0,Y 361.952,Z 160.878,A -85,B 0,C 180,E1 -13113.474,E2 -13113.474} C_VEL
LIN {X 0,Y 361.891,Z 160.906,A -85,B 0,C 180,E1 -13117.144,E2 -13117.144} C_VEL
LIN {X 0,Y 361.905,Z 160.879,A -85,B 0,C 180,E1 -13120.723,E2 -13120.723} C_VEL
LIN {X 0,Y 361.931,Z 160.886,A -85,B 0,C 180,E1 -13123.065,E2 -13123.065} C_VEL
LIN {X 0,Y 361.997,Z 160.893,A -85,B 0,C 180,E1 -13126.527,E2 -13126.527} C_VEL
LIN {X 0,Y 362.028,Z 160.861,A -85,B 0,C 180,E1 -13129.937,E2 -13129.937} C_VEL
LIN {X 0,Y 362.162,Z 160.867,A -85,B 0,C 180,E1 -13133.313,E2 -13133.313} C_VEL
LIN {X 0,Y 362.278,Z 160.85,A -85,B 0,C 180,E1 -13137.776,E2 -13137.776} C_VEL
LIN {X 0,Y 362.423,Z 160.81,A -85,B 0,C 180,E1 -13139.999,E2 -13139.999} C_VEL
LIN {X 0,Y 362.279,Z 160.842,A -85,B 0,C 180,E1 -13142.223,E2 -13142.223} C_VEL
LIN {X 0,Y 362.168,Z 160.865,A -85,B 0,C 180,E1 -13146.686,E2 -13146.686} C_VEL
LIN {X 0,Y 362.07,Z 160.859,A -85,B 0,C 180,E1 -13148.933,E2 -13148.933} C_VEL
LIN {X 0,Y 361.956,Z 160.889,A -85,B 0,C 180,E1 -13152.332,E2 -13152.332} C_VEL
LIN {X 0,Y 361.958,Z 160.896,A -85,B 0,C 180,E1 -13154.62,E2 -13154.62} C_VEL
LIN {X 0,Y 361.952,Z 160.875,A -85,B 0,C 180,E1 -13158.099,E2 -13158.099} C_VEL
LIN {X 0,Y 361.888,Z 160.9,A -85,B 0,C 180,E1 -13161.652,E2 -13161.652} C_VEL
LIN {X 0,Y 361.924,Z 160.897,A -85,B 0,C 180,E1 -13165.29,E2 -13165.29} C_VEL
LIN {X 0,Y 361.918,Z 160.884,A -85,B 0,C 180,E1 -13167.777,E2 -13167.777} C_VEL
LIN {X 0,Y 361.842,Z 160.914,A -85,B 0,C 180,E1 -13171.285,E2 -13171.285} C_VEL
LIN {X 0,Y 361.85,Z 160.891,A -85,B 0,C 180,E1 -13174.28,E2 -13174.28} C_VEL
LIN {X 0,Y 361.866,Z 160.91,A -85,B 0,C 180,E1 -13177.224,E2 -13177.224} C_VEL
LIN {X 0,Y 361.831,Z 160.9,A -85,B 0,C 180,E1 -13180.755,E2 -13180.755} C_VEL
LIN {X 0,Y 361.831,Z 160.911,A -85,B 0,C 180,E1 -13184.365,E2 -13184.365} C_VEL
LIN {X 0,Y 361.831,Z 160.87,A -85,B 0,C 180,E1 -13187.568,E2 -13187.568} C_VEL
LIN {X 0,Y 361.867,Z 160.911,A -85,B 0,C 180,E1 -13191.576,E2 -13191.576} C_VEL
LIN {X 0,Y 361.87,Z 160.885,A -85,B 0,C 180,E1 -13194.655,E2 -13194.655} C_VEL
LIN {X 0,Y 361.857,Z 160.912,A -85,B 0,C 180,E1 -13198.373,E2 -13198.373} C_VEL
LIN {X 0,Y 361.918,Z 160.9,A -85,B 0,C 180,E1 -13202.222,E2 -13202.222} C_VEL
LIN {X 0,Y 361.924,Z 160.904,A -85,B 0,C 180,E1 -13204.71,E2 -13204.71} C_VEL
LIN {X 0,Y 361.888,Z 160.909,A -85,B 0,C 180,E1 -13208.347,E2 -13208.347} C_VEL
LIN {X 0,Y 361.959,Z 161.006,A -85,B 0,C 180,E1 -13212.141,E2 -13212.141} C_VEL
LIN {X 0,Y 362.155,Z 161.988,A -85,B 0,C 180,E1 -13212.51,E2 -13212.51} C_VEL
LIN {X 0,Y 363.707,Z 164.762,A -85,B 0,C 180,E1 -13213.03,E2 -13213.03} C_VEL
LIN {X 0,Y 366.072,Z 166.534,A -85,B 0,C 180,E1 -13213.721,E2 -13213.721} C_VEL
LIN {X 0,Y 368.394,Z 169.962,A -85,B 0,C 180,E1 -13214.47,E2 -13214.47} C_VEL
LIN {X 0,Y 371.016,Z 172.152,A -85,B 0,C 180,E1 -13215.324,E2 -13215.324} C_VEL
LIN {X 0,Y 371.855,Z 172.829,A -85,B 0,C 180,E1 -13215.602,E2 -13215.602} C_VEL
LIN {X 0,Y 374.176,Z 176.038,A -85,B 0,C 180,E1 -13216.445,E2 -13216.445} C_VEL
LIN {X 0,Y 376.963,Z 178.261,A -85,B 0,C 180,E1 -13217.483,E2 -13217.483} C_VEL
LIN {X 0,Y 377.933,Z 179.025,A -85,B 0,C 180,E1 -13217.856,E2 -13217.856} C_VEL
LIN {X 0,Y 380.359,Z 182.21,A -85,B 0,C 180,E1 -13218.948,E2 -13218.948} C_VEL
LIN {X 0,Y 383.085,Z 184.368,A -85,B 0,C 180,E1 -13220.237,E2 -13220.237} C_VEL
LIN {X 0,Y 384.988,Z 185.447,A -85,B 0,C 180,E1 -13221.206,E2 -13221.206} C_VEL
LIN {X 0,Y 387.164,Z 188.427,A -85,B 0,C 180,E1 -13222.596,E2 -13222.596} C_VEL
LIN {X 0,Y 389.397,Z 190.369,A -85,B 0,C 180,E1 -13224.303,E2 -13224.303} C_VEL
LIN {X 0,Y 391.009,Z 191.291,A -85,B 0,C 180,E1 -13225.877,E2 -13225.877} C_VEL
LIN {X 0,Y 392.127,Z 191.663,A -85,B 0,C 180,E1 -13227.451,E2 -13227.451} C_VEL
LIN {X 0,Y 392.685,Z 192.085,A -85,B 0,C 180,E1 -13228.975,E2 -13228.975} C_VEL
LIN {X 0,Y 392.864,Z 192.021,A -85,B 0,C 180,E1 -13230,E2 -13230} C_VEL
LIN {X 0,Y 392.598,Z 191.97,A -85,B 0,C 180,E1 -13231.539,E2 -13231.539} C_VEL
LIN {X 0,Y 391.864,Z 191.541,A -85,B 0,C 180,E1 -13233.084,E2 -13233.084} C_VEL
LIN {X 0,Y 390.285,Z 190.93,A -85,B 0,C 180,E1 -13234.907,E2 -13234.907} C_VEL
LIN {X 0,Y 388.217,Z 189.445,A -85,B 0,C 180,E1 -13236.635,E2 -13236.635} C_VEL
LIN {X 0,Y 386.33,Z 187.398,A -85,B 0,C 180,E1 -13237.961,E2 -13237.961} C_VEL
LIN {X 0,Y 384.776,Z 185.128,A -85,B 0,C 180,E1 -13238.931,E2 -13238.931} C_VEL
LIN {X 0,Y 381.795,Z 183.489,A -85,B 0,C 180,E1 -13240.39,E2 -13240.39} C_VEL
LIN {X 0,Y 379.034,Z 180.744,A -85,B 0,C 180,E1 -13241.628,E2 -13241.628} C_VEL
LIN {X 0,Y 377.387,Z 178.465,A -85,B 0,C 180,E1 -13242.366,E2 -13242.366} C_VEL
LIN {X 0,Y 374.536,Z 176.421,A -85,B 0,C 180,E1 -13243.414,E2 -13243.414} C_VEL
LIN {X 0,Y 372.157,Z 173.346,A -85,B 0,C 180,E1 -13244.288,E2 -13244.288} C_VEL
LIN {X 0,Y 371.417,Z 172.369,A -85,B 0,C 180,E1 -13244.548,E2 -13244.548} C_VEL
LIN {X 0,Y 368.752,Z 170.355,A -85,B 0,C 180,E1 -13245.422,E2 -13245.422} C_VEL
LIN {X 0,Y 366.726,Z 167.567,A -85,B 0,C 180,E1 -13246.063,E2 -13246.063} C_VEL
LIN {X 0,Y 366.071,Z 166.534,A -85,B 0,C 180,E1 -13246.279,E2 -13246.279} C_VEL
LIN {X 0,Y 363.707,Z 164.762,A -85,B 0,C 180,E1 -13246.97,E2 -13246.97} C_VEL
LIN {X 0,Y 362.199,Z 162.119,A -85,B 0,C 180,E1 -13247.466,E2 -13247.466} C_VEL
LIN {X 0,Y 361.973,Z 161.105,A -85,B 0,C 180,E1 -13247.778,E2 -13247.778} C_VEL
LIN {X 0,Y 361.88,Z 160.91,A -85,B 0,C 180,E1 -13251.222,E2 -13251.222} C_VEL
LIN {X 0,Y 361.891,Z 160.907,A -85,B 0,C 180,E1 -13254.114,E2 -13254.114} C_VEL
LIN {X 0,Y 361.939,Z 160.902,A -85,B 0,C 180,E1 -13256.722,E2 -13256.722} C_VEL
LIN {X 0,Y 361.872,Z 160.898,A -85,B 0,C 180,E1 -13260.328,E2 -13260.328} C_VEL
LIN {X 0,Y 361.852,Z 160.885,A -85,B 0,C 180,E1 -13264.28,E2 -13264.28} C_VEL
LIN {X 0,Y 361.866,Z 160.909,A -85,B 0,C 180,E1 -13267.225,E2 -13267.225} C_VEL
LIN {X 0,Y 361.83,Z 160.881,A -85,B 0,C 180,E1 -13270.755,E2 -13270.755} C_VEL
LIN {X 0,Y 361.831,Z 160.897,A -85,B 0,C 180,E1 -13274.366,E2 -13274.366} C_VEL
LIN {X 0,Y 361.832,Z 160.91,A -85,B 0,C 180,E1 -13277.568,E2 -13277.568} C_VEL
LIN {X 0,Y 361.828,Z 160.9,A -85,B 0,C 180,E1 -13279.589,E2 -13279.589} C_VEL
LIN {X 0,Y 361.18,Z 160.988,A -85,B 0,C 180,E1 -13280.518,E2 -13280.518} C_VEL
LIN {X 0,Y 358.351,Z 161.347,A -85,B 0,C 180,E1 -13282.029,E2 -13282.029} C_VEL
LIN {X 0,Y 355.941,Z 161.646,A -85,B 0,C 180,E1 -13283.251,E2 -13283.251} C_VEL
LIN {X 0,Y 354.898,Z 161.769,A -85,B 0,C 180,E1 -13284.197,E2 -13284.197} C_VEL
LIN {X 0,Y 354.809,Z 161.775,A -85,B 0,C 180,E1 -13284.517,E2 -13284.517} C_VEL
LIN {X 0,Y 354.782,Z 161.787,A -85,B 0,C 180,E1 -13287.667,E2 -13287.667} C_VEL
LIN {X 0,Y 354.864,Z 161.774,A -85,B 0,C 180,E1 -13290.622,E2 -13290.622} C_VEL
LIN {X 0,Y 354.895,Z 161.764,A -85,B 0,C 180,E1 -13294.173,E2 -13294.173} C_VEL
LIN {X 0,Y 354.83,Z 161.785,A -85,B 0,C 180,E1 -13297.894,E2 -13297.894} C_VEL
LIN {X 0,Y 354.918,Z 161.75,A -85,B 0,C 180,E1 -13301.892,E2 -13301.892} C_VEL
LIN {X 0,Y 354.939,Z 161.773,A -85,B 0,C 180,E1 -13305.982,E2 -13305.982} C_VEL
LIN {X 0,Y 354.974,Z 161.739,A -85,B 0,C 180,E1 -13309.736,E2 -13309.736} C_VEL
LIN {X 0,Y 355.125,Z 161.733,A -85,B 0,C 180,E1 -13312.038,E2 -13312.038} C_VEL
LIN {X 0,Y 355.089,Z 161.752,A -85,B 0,C 180,E1 -13314.321,E2 -13314.321} C_VEL
LIN {X 0,Y 355.242,Z 161.719,A -85,B 0,C 180,E1 -13317.733,E2 -13317.733} C_VEL
LIN {X 0,Y 355.371,Z 161.688,A -85,B 0,C 180,E1 -13320.001,E2 -13320.001} C_VEL
LIN {X 0,Y 355.241,Z 161.726,A -85,B 0,C 180,E1 -13322.268,E2 -13322.268} C_VEL
LIN {X 0,Y 355.125,Z 161.744,A -85,B 0,C 180,E1 -13326.82,E2 -13326.82} C_VEL
LIN {X 0,Y 354.975,Z 161.74,A -85,B 0,C 180,E1 -13330.265,E2 -13330.265} C_VEL
LIN {X 0,Y 354.94,Z 161.768,A -85,B 0,C 180,E1 -13334.019,E2 -13334.019} C_VEL
LIN {X 0,Y 354.921,Z 161.748,A -85,B 0,C 180,E1 -13338.109,E2 -13338.109} C_VEL
LIN {X 0,Y 354.835,Z 161.78,A -85,B 0,C 180,E1 -13342.107,E2 -13342.107} C_VEL
LIN {X 0,Y 354.898,Z 161.761,A -85,B 0,C 180,E1 -13345.828,E2 -13345.828} C_VEL
LIN {X 0,Y 354.817,Z 161.784,A -85,B 0,C 180,E1 -13349.683,E2 -13349.683} C_VEL
LIN {X 0,Y 354.806,Z 161.772,A -85,B 0,C 180,E1 -13353.703,E2 -13353.703} C_VEL
LIN {X 0,Y 354.797,Z 161.787,A -85,B 0,C 180,E1 -13356.46,E2 -13356.46} C_VEL
LIN {X 0,Y 354.824,Z 161.776,A -85,B 0,C 180,E1 -13359.424,E2 -13359.424} C_VEL
LIN {X 0,Y 354.788,Z 161.79,A -85,B 0,C 180,E1 -13362.868,E2 -13362.868} C_VEL
LIN {X 0,Y 354.768,Z 161.793,A -85,B 0,C 180,E1 -13366.104,E2 -13366.104} C_VEL
LIN {X 0,Y 354.788,Z 161.769,A -85,B 0,C 180,E1 -13369.18,E2 -13369.18} C_VEL
LIN {X 0,Y 354.813,Z 161.79,A -85,B 0,C 180,E1 -13372.402,E2 -13372.402} C_VEL
LIN {X 0,Y 354.813,Z 161.774,A -85,B 0,C 180,E1 -13374.941,E2 -13374.941} C_VEL
LIN {X 0,Y 354.881,Z 161.947,A -85,B 0,C 180,E1 -13378.082,E2 -13378.082} C_VEL
LIN {X 0,Y 356.41,Z 169.546,A -85,B 0,C 180,E1 -13380.788,E2 -13380.788} C_VEL
LIN {X 0,Y 357.924,Z 177.913,A -85,B 0,C 180,E1 -13383.468,E2 -13383.468} C_VEL
LIN {X 0,Y 357.815,Z 181.667,A -85,B 0,C 180,E1 -13384.624,E2 -13384.624} C_VEL
LIN {X 0,Y 356.79,Z 190.803,A -85,B 0,C 180,E1 -13387.392,E2 -13387.392} C_VEL
LIN {X 0,Y 357.93,Z 196.382,A -85,B 0,C 180,E1 -13387.637,E2 -13387.637} C_VEL
LIN {X 0,Y 362.831,Z 222.262,A -85,B 0,C 180,E1 -13388.492,E2 -13388.492} C_VEL
LIN {X 0,Y 363.534,Z 226.985,A -85,B 0,C 180,E1 -13388.633,E2 -13388.633} C_VEL
LIN {X 0,Y 362.33,Z 295.608,A -85,B 0,C 180,E1 -13390.01,E2 -13390.01} C_VEL
LIN {X 0,Y 361.914,Z 305.493,A -85,B 0,C 180,E1 -13390.318,E2 -13390.318} C_VEL
LIN {X 0,Y 361.264,Z 315.466,A -85,B 0,C 180,E1 -13390.762,E2 -13390.762} C_VEL
LIN {X 0,Y 360.476,Z 325.827,A -85,B 0,C 180,E1 -13391.382,E2 -13391.382} C_VEL
LIN {X 0,Y 359.656,Z 334.96,A -85,B 0,C 180,E1 -13392.075,E2 -13392.075} C_VEL
LIN {X 0,Y 358.708,Z 343.954,A -85,B 0,C 180,E1 -13392.909,E2 -13392.909} C_VEL
LIN {X 0,Y 357.75,Z 352.682,A -85,B 0,C 180,E1 -13393.89,E2 -13393.89} C_VEL
LIN {X 0,Y 356.943,Z 360.393,A -85,B 0,C 180,E1 -13394.926,E2 -13394.926} C_VEL
LIN {X 0,Y 356.212,Z 367.299,A -85,B 0,C 180,E1 -13396.014,E2 -13396.014} C_VEL
LIN {X 0,Y 355.478,Z 373.5,A -85,B 0,C 180,E1 -13397.149,E2 -13397.149} C_VEL
LIN {X 0,Y 354.667,Z 380.035,A -85,B 0,C 180,E1 -13398.571,E2 -13398.571} C_VEL
LIN {X 0,Y 354.248,Z 384.539,A -85,B 0,C 180,E1 -13399.715,E2 -13399.715} C_VEL
LIN {X 0,Y 353.726,Z 390.03,A -85,B 0,C 180,E1 -13401.43,E2 -13401.43} C_VEL
LIN {X 0,Y 353.418,Z 394.356,A -85,B 0,C 180,E1 -13403.148,E2 -13403.148} C_VEL
LIN {X 0,Y 353.291,Z 396.723,A -85,B 0,C 180,E1 -13404.292,E2 -13404.292} C_VEL
LIN {X 0,Y 353.263,Z 398.523,A -85,B 0,C 180,E1 -13405.436,E2 -13405.436} C_VEL
LIN {X 0,Y 353.172,Z 400.967,A -85,B 0,C 180,E1 -13407.719,E2 -13407.719} C_VEL
LIN {X 0,Y 353.204,Z 401.557,A -85,B 0,C 180,E1 -13408.86,E2 -13408.86} C_VEL
LIN {X 0,Y 353.204,Z 401.557,A -85,B 0,C 180,E1 -13411.14,E2 -13411.14} C_VEL
LIN {X 0,Y 353.172,Z 400.967,A -85,B 0,C 180,E1 -13412.281,E2 -13412.281} C_VEL
LIN {X 0,Y 353.263,Z 398.523,A -85,B 0,C 180,E1 -13414.564,E2 -13414.564} C_VEL
LIN {X 0,Y 353.298,Z 396.301,A -85,B 0,C 180,E1 -13415.937,E2 -13415.937} C_VEL
LIN {X 0,Y 353.514,Z 393.116,A -85,B 0,C 180,E1 -13417.425,E2 -13417.425} C_VEL
LIN {X 0,Y 353.877,Z 388.37,A -85,B 0,C 180,E1 -13419.142,E2 -13419.142} C_VEL
LIN {X 0,Y 354.456,Z 382.348,A -85,B 0,C 180,E1 -13420.857,E2 -13420.857} C_VEL
LIN {X 0,Y 355.139,Z 376.252,A -85,B 0,C 180,E1 -13422.283,E2 -13422.283} C_VEL
LIN {X 0,Y 355.854,Z 370.553,A -85,B 0,C 180,E1 -13423.418,E2 -13423.418} C_VEL
LIN {X 0,Y 356.8,Z 361.998,A -85,B 0,C 180,E1 -13424.837,E2 -13424.837} C_VEL
LIN {X 0,Y 357.669,Z 353.817,A -85,B 0,C 180,E1 -13425.967,E2 -13425.967} C_VEL
LIN {X 0,Y 358.554,Z 345.305,A -85,B 0,C 180,E1 -13426.951,E2 -13426.951} C_VEL
LIN {X 0,Y 359.474,Z 336.591,A -85,B 0,C 180,E1 -13427.787,E2 -13427.787} C_VEL
LIN {X 0,Y 360.379,Z 326.834,A -85,B 0,C 180,E1 -13428.549,E2 -13428.549} C_VEL
LIN {X 0,Y 361.187,Z 316.754,A -85,B 0,C 180,E1 -13429.169,E2 -13429.169} C_VEL
LIN {X 0,Y 361.78,Z 307.24,A -85,B 0,C 180,E1 -13429.615,E2 -13429.615} C_VEL
LIN {X 0,Y 362.296,Z 296.931,A -85,B 0,C 180,E1 -13429.955,E2 -13429.955} C_VEL
LIN {X 0,Y 363.358,Z 240.629,A -85,B 0,C 180,E1 -13431.094,E2 -13431.094} C_VEL
LIN {X 0,Y 363.306,Z 225.337,A -85,B 0,C 180,E1 -13431.415,E2 -13431.415} C_VEL
LIN {X 0,Y 358.441,Z 198.906,A -85,B 0,C 180,E1 -13432.276,E2 -13432.276} C_VEL
LIN {X 0,Y 356.787,Z 191.088,A -85,B 0,C 180,E1 -13432.577,E2 -13432.577} C_VEL
LIN {X 0,Y 356.835,Z 189.646,A -85,B 0,C 180,E1 -13432.899,E2 -13432.899} C_VEL
LIN {X 0,Y 357.946,Z 180.961,A -85,B 0,C 180,E1 -13435.591,E2 -13435.591} C_VEL
LIN {X 0,Y 357.825,Z 176.967,A -85,B 0,C 180,E1 -13436.855,E2 -13436.855} C_VEL
LIN {X 0,Y 356.171,Z 168.253,A -85,B 0,C 180,E1 -13439.747,E2 -13439.747} C_VEL
LIN {X 0,Y 354.861,Z 161.845,A -85,B 0,C 180,E1 -13441.971,E2 -13441.971} C_VEL
LIN {X 0,Y 354.823,Z 161.773,A -85,B 0,C 180,E1 -13445.699,E2 -13445.699} C_VEL
LIN {X 0,Y 354.825,Z 161.767,A -85,B 0,C 180,E1 -13449.423,E2 -13449.423} C_VEL
LIN {X 0,Y 354.789,Z 161.79,A -85,B 0,C 180,E1 -13452.867,E2 -13452.867} C_VEL
LIN {X 0,Y 354.767,Z 161.791,A -85,B 0,C 180,E1 -13456.103,E2 -13456.103} C_VEL
LIN {X 0,Y 354.787,Z 161.784,A -85,B 0,C 180,E1 -13459.178,E2 -13459.178} C_VEL
LIN {X 0,Y 354.806,Z 161.787,A -85,B 0,C 180,E1 -13462.402,E2 -13462.402} C_VEL
LIN {X 0,Y 354.811,Z 161.775,A -85,B 0,C 180,E1 -13464.94,E2 -13464.94} C_VEL
LIN {X 0,Y 354.792,Z 161.787,A -85,B 0,C 180,E1 -13468.405,E2 -13468.405} C_VEL
LIN {X 0,Y 354.845,Z 161.77,A -85,B 0,C 180,E1 -13471.618,E2 -13471.618} C_VEL
LIN {X 0,Y 354.898,Z 161.761,A -85,B 0,C 180,E1 -13474.172,E2 -13474.172} C_VEL
LIN {X 0,Y 354.835,Z 161.78,A -85,B 0,C 180,E1 -13477.893,E2 -13477.893} C_VEL
LIN {X 0,Y 354.921,Z 161.748,A -85,B 0,C 180,E1 -13481.891,E2 -13481.891} C_VEL
LIN {X 0,Y 354.94,Z 161.768,A -85,B 0,C 180,E1 -13485.981,E2 -13485.981} C_VEL
LIN {X 0,Y 354.975,Z 161.74,A -85,B 0,C 180,E1 -13489.735,E2 -13489.735} C_VEL
LIN {X 0,Y 355.125,Z 161.744,A -85,B 0,C 180,E1 -13493.18,E2 -13493.18} C_VEL
LIN {X 0,Y 355.241,Z 161.726,A -85,B 0,C 180,E1 -13497.732,E2 -13497.732} C_VEL
LIN {X 0,Y 355.371,Z 161.688,A -85,B 0,C 180,E1 -13499.999,E2 -13499.999} C_VEL
LIN {X 0,Y 355.242,Z 161.719,A -85,B 0,C 180,E1 -13502.267,E2 -13502.267} C_VEL
LIN {X 0,Y 355.134,Z 161.74,A -85,B 0,C 180,E1 -13506.819,E2 -13506.819} C_VEL
LIN {X 0,Y 355.012,Z 161.737,A -85,B 0,C 180,E1 -13509.112,E2 -13509.112} C_VEL
LIN {X 0,Y 354.917,Z 161.77,A -85,B 0,C 180,E1 -13512.58,E2 -13512.58} C_VEL
LIN {X 0,Y 354.885,Z 161.774,A -85,B 0,C 180,E1 -13516.095,E2 -13516.095} C_VEL
LIN {X 0,Y 354.897,Z 161.75,A -85,B 0,C 180,E1 -13518.472,E2 -13518.472} C_VEL
LIN {X 0,Y 354.83,Z 161.785,A -85,B 0,C 180,E1 -13522.106,E2 -13522.106} C_VEL
LIN {X 0,Y 354.895,Z 161.764,A -85,B 0,C 180,E1 -13525.827,E2 -13525.827} C_VEL
LIN {X 0,Y 354.85,Z 161.779,A -85,B 0,C 180,E1 -13529.678,E2 -13529.678} C_VEL
LIN {X 0,Y 354.801,Z 161.773,A -85,B 0,C 180,E1 -13533.702,E2 -13533.702} C_VEL
LIN {X 0,Y 354.797,Z 161.786,A -85,B 0,C 180,E1 -13536.459,E2 -13536.459} C_VEL
LIN {X 0,Y 354.819,Z 161.779,A -85,B 0,C 180,E1 -13539.423,E2 -13539.423} C_VEL
LIN {X 0,Y 354.784,Z 161.79,A -85,B 0,C 180,E1 -13542.867,E2 -13542.867} C_VEL
LIN {X 0,Y 354.772,Z 161.77,A -85,B 0,C 180,E1 -13546.105,E2 -13546.105} C_VEL
LIN {X 0,Y 354.782,Z 161.757,A -85,B 0,C 180,E1 -13549.179,E2 -13549.179} C_VEL
LIN {X 0,Y 354.807,Z 161.79,A -85,B 0,C 180,E1 -13552.401,E2 -13552.401} C_VEL
LIN {X 0,Y 354.808,Z 161.762,A -85,B 0,C 180,E1 -13554.941,E2 -13554.941} C_VEL
LIN {X 0,Y 354.812,Z 161.79,A -85,B 0,C 180,E1 -13558.399,E2 -13558.399} C_VEL
LIN {X 0,Y 354.85,Z 161.77,A -85,B 0,C 180,E1 -13561.619,E2 -13561.619} C_VEL
LIN {X 0,Y 354.895,Z 161.779,A -85,B 0,C 180,E1 -13564.173,E2 -13564.173} C_VEL
LIN {X 0,Y 354.831,Z 161.788,A -85,B 0,C 180,E1 -13567.894,E2 -13567.894} C_VEL
LIN {X 0,Y 354.913,Z 162.031,A -85,B 0,C 180,E1 -13570.667,E2 -13570.667} C_VEL
LIN {X 0,Y 355.229,Z 163.267,A -85,B 0,C 180,E1 -13570.97,E2 -13570.97} C_VEL
LIN {X 0,Y 356.801,Z 165.799,A -85,B 0,C 180,E1 -13571.427,E2 -13571.427} C_VEL
LIN {X 0,Y 359.108,Z 167.687,A -85,B 0,C 180,E1 -13572.017,E2 -13572.017} C_VEL
LIN {X 0,Y 361.33,Z 171.095,A -85,B 0,C 180,E1 -13572.684,E2 -13572.684} C_VEL
LIN {X 0,Y 364.119,Z 173.437,A -85,B 0,C 180,E1 -13573.452,E2 -13573.452} C_VEL
LIN {X 0,Y 366.534,Z 176.728,A -85,B 0,C 180,E1 -13574.233,E2 -13574.233} C_VEL
LIN {X 0,Y 370,Z 179.608,A -85,B 0,C 180,E1 -13575.326,E2 -13575.326} C_VEL
LIN {X 0,Y 372.698,Z 182.952,A -85,B 0,C 180,E1 -13576.266,E2 -13576.266} C_VEL
LIN {X 0,Y 376.196,Z 185.696,A -85,B 0,C 180,E1 -13577.56,E2 -13577.56} C_VEL
LIN {X 0,Y 378.902,Z 188.996,A -85,B 0,C 180,E1 -13578.736,E2 -13578.736} C_VEL
LIN {X 0,Y 381.523,Z 191.073,A -85,B 0,C 180,E1 -13579.928,E2 -13579.928} C_VEL
LIN {X 0,Y 383.693,Z 192.297,A -85,B 0,C 180,E1 -13580.976,E2 -13580.976} C_VEL
LIN {X 0,Y 386.239,Z 195.581,A -85,B 0,C 180,E1 -13582.578,E2 -13582.578} C_VEL
LIN {X 0,Y 388.48,Z 197.392,A -85,B 0,C 180,E1 -13584.264,E2 -13584.264} C_VEL
LIN {X 0,Y 390.134,Z 198.331,A -85,B 0,C 180,E1 -13585.868,E2 -13585.868} C_VEL
LIN {X 0,Y 391.261,Z 198.71,A -85,B 0,C 180,E1 -13587.445,E2 -13587.445} C_VEL
LIN {X 0,Y 391.823,Z 199.131,A -85,B 0,C 180,E1 -13588.972,E2 -13588.972} C_VEL
LIN {X 0,Y 391.999,Z 199.068,A -85,B 0,C 180,E1 -13590,E2 -13590} C_VEL
LIN {X 0,Y 391.73,Z 199.017,A -85,B 0,C 180,E1 -13591.542,E2 -13591.542} C_VEL
LIN {X 0,Y 390.988,Z 198.587,A -85,B 0,C 180,E1 -13593.091,E2 -13593.091} C_VEL
LIN {X 0,Y 389.394,Z 197.974,A -85,B 0,C 180,E1 -13594.918,E2 -13594.918} C_VEL
LIN {X 0,Y 387.301,Z 196.534,A -85,B 0,C 180,E1 -13596.652,E2 -13596.652} C_VEL
LIN {X 0,Y 385.37,Z 194.628,A -85,B 0,C 180,E1 -13597.981,E2 -13597.981} C_VEL
LIN {X 0,Y 383.438,Z 192.006,A -85,B 0,C 180,E1 -13599.167,E2 -13599.167} C_VEL
LIN {X 0,Y 380.179,Z 190.111,A -85,B 0,C 180,E1 -13600.72,E2 -13600.72} C_VEL
LIN {X 0,Y 377.084,Z 186.94,A -85,B 0,C 180,E1 -13602.069,E2 -13602.069} C_VEL
LIN {X 0,Y 375.688,Z 185.212,A -85,B 0,C 180,E1 -13602.629,E2 -13602.629} C_VEL
LIN {X 0,Y 372.662,Z 182.89,A -85,B 0,C 180,E1 -13603.749,E2 -13603.749} C_VEL
LIN {X 0,Y 369.993,Z 179.655,A -85,B 0,C 180,E1 -13604.675,E2 -13604.675} C_VEL
LIN {X 0,Y 368.754,Z 178.5,A -85,B 0,C 180,E1 -13605.1,E2 -13605.1} C_VEL
LIN {X 0,Y 365.639,Z 175.729,A -85,B 0,C 180,E1 -13606.045,E2 -13606.045} C_VEL
LIN {X 0,Y 363.644,Z 172.895,A -85,B 0,C 180,E1 -13606.693,E2 -13606.693} C_VEL
LIN {X 0,Y 360.934,Z 170.672,A -85,B 0,C 180,E1 -13607.427,E2 -13607.427} C_VEL
LIN {X 0,Y 358.716,Z 167.217,A -85,B 0,C 180,E1 -13608.097,E2 -13608.097} C_VEL
LIN {X 0,Y 356.497,Z 165.479,A -85,B 0,C 180,E1 -13608.649,E2 -13608.649} C_VEL
LIN {X 0,Y 355.027,Z 162.604,A -85,B 0,C 180,E1 -13609.14,E2 -13609.14} C_VEL
LIN {X 0,Y 354.86,Z 161.836,A -85,B 0,C 180,E1 -13609.524,E2 -13609.524} C_VEL
LIN {X 0,Y 354.828,Z 161.789,A -85,B 0,C 180,E1 -13613.337,E2 -13613.337} C_VEL
LIN {X 0,Y 354.885,Z 161.781,A -85,B 0,C 180,E1 -13616.982,E2 -13616.982} C_VEL
LIN {X 0,Y 354.85,Z 161.766,A -85,B 0,C 180,E1 -13619.679,E2 -13619.679} C_VEL
LIN {X 0,Y 354.826,Z 161.765,A -85,B 0,C 180,E1 -13623.682,E2 -13623.682} C_VEL
LIN {X 0,Y 354.797,Z 161.781,A -85,B 0,C 180,E1 -13626.459,E2 -13626.459} C_VEL
LIN {X 0,Y 354.819,Z 161.778,A -85,B 0,C 180,E1 -13629.424,E2 -13629.424} C_VEL
LIN {X 0,Y 354.783,Z 161.751,A -85,B 0,C 180,E1 -13632.867,E2 -13632.867} C_VEL
LIN {X 0,Y 354.772,Z 161.791,A -85,B 0,C 180,E1 -13636.105,E2 -13636.105} C_VEL
LIN {X 0,Y 354.772,Z 161.778,A -85,B 0,C 180,E1 -13639.588,E2 -13639.588} C_VEL
LIN {X 0,Y 354.807,Z 161.791,A -85,B 0,C 180,E1 -13642.402,E2 -13642.402} C_VEL
LIN {X 0,Y 354.809,Z 161.775,A -85,B 0,C 180,E1 -13644.517,E2 -13644.517} C_VEL
LIN {X 0,Y 354.118,Z 161.857,A -85,B 0,C 180,E1 -13645.464,E2 -13645.464} C_VEL
LIN {X 0,Y 351.223,Z 162.229,A -85,B 0,C 180,E1 -13647.004,E2 -13647.004} C_VEL
LIN {X 0,Y 348.807,Z 162.536,A -85,B 0,C 180,E1 -13648.25,E2 -13648.25} C_VEL
LIN {X 0,Y 347.811,Z 162.659,A -85,B 0,C 180,E1 -13649.214,E2 -13649.214} C_VEL
LIN {X 0,Y 347.751,Z 162.666,A -85,B 0,C 180,E1 -13649.541,E2 -13649.541} C_VEL
LIN {X 0,Y 347.848,Z 162.633,A -85,B 0,C 180,E1 -13652.745,E2 -13652.745} C_VEL
LIN {X 0,Y 347.784,Z 162.664,A -85,B 0,C 180,E1 -13656.162,E2 -13656.162} C_VEL
LIN {X 0,Y 347.808,Z 162.638,A -85,B 0,C 180,E1 -13659.91,E2 -13659.91} C_VEL
LIN {X 0,Y 347.862,Z 162.635,A -85,B 0,C 180,E1 -13662.36,E2 -13662.36} C_VEL
LIN {X 0,Y 347.894,Z 162.651,A -85,B 0,C 180,E1 -13665.971,E2 -13665.971} C_VEL
LIN {X 0,Y 347.925,Z 162.618,A -85,B 0,C 180,E1 -13669.526,E2 -13669.526} C_VEL
LIN {X 0,Y 348.104,Z 162.615,A -85,B 0,C 180,E1 -13673.043,E2 -13673.043} C_VEL
LIN {X 0,Y 348.205,Z 162.595,A -85,B 0,C 180,E1 -13677.687,E2 -13677.687} C_VEL
LIN {X 0,Y 348.322,Z 162.565,A -85,B 0,C 180,E1 -13680.001,E2 -13680.001} C_VEL
LIN {X 0,Y 348.203,Z 162.603,A -85,B 0,C 180,E1 -13682.314,E2 -13682.314} C_VEL
LIN {X 0,Y 348.09,Z 162.618,A -85,B 0,C 180,E1 -13686.959,E2 -13686.959} C_VEL
LIN {X 0,Y 347.926,Z 162.619,A -85,B 0,C 180,E1 -13690.475,E2 -13690.475} C_VEL
LIN {X 0,Y 347.897,Z 162.645,A -85,B 0,C 180,E1 -13694.151,E2 -13694.151} C_VEL
LIN {X 0,Y 347.889,Z 162.622,A -85,B 0,C 180,E1 -13698.291,E2 -13698.291} C_VEL
LIN {X 0,Y 347.789,Z 162.659,A -85,B 0,C 180,E1 -13701.636,E2 -13701.636} C_VEL
LIN {X 0,Y 347.811,Z 162.648,A -85,B 0,C 180,E1 -13705.109,E2 -13705.109} C_VEL
LIN {X 0,Y 347.807,Z 162.642,A -85,B 0,C 180,E1 -13707.695,E2 -13707.695} C_VEL
LIN {X 0,Y 347.748,Z 162.667,A -85,B 0,C 180,E1 -13710.349,E2 -13710.349} C_VEL
LIN {X 0,Y 347.748,Z 162.649,A -85,B 0,C 180,E1 -13714.045,E2 -13714.045} C_VEL
LIN {X 0,Y 347.761,Z 162.665,A -85,B 0,C 180,E1 -13717.322,E2 -13717.322} C_VEL
LIN {X 0,Y 347.732,Z 162.658,A -85,B 0,C 180,E1 -13720.298,E2 -13720.298} C_VEL
LIN {X 0,Y 347.723,Z 162.668,A -85,B 0,C 180,E1 -13723.409,E2 -13723.409} C_VEL
LIN {X 0,Y 347.726,Z 162.672,A -85,B 0,C 180,E1 -13726.687,E2 -13726.687} C_VEL
LIN {X 0,Y 347.748,Z 162.644,A -85,B 0,C 180,E1 -13730.174,E2 -13730.174} C_VEL
LIN {X 0,Y 347.767,Z 162.665,A -85,B 0,C 180,E1 -13732.68,E2 -13732.68} C_VEL
LIN {X 0,Y 347.75,Z 162.666,A -85,B 0,C 180,E1 -13735.957,E2 -13735.957} C_VEL
LIN {X 0,Y 347.818,Z 162.801,A -85,B 0,C 180,E1 -13737.704,E2 -13737.704} C_VEL
LIN {X 0,Y 349.426,Z 170.703,A -85,B 0,C 180,E1 -13740.57,E2 -13740.57} C_VEL
LIN {X 0,Y 350.937,Z 178.779,A -85,B 0,C 180,E1 -13743.219,E2 -13743.219} C_VEL
LIN {X 0,Y 350.906,Z 182.209,A -85,B 0,C 180,E1 -13744.326,E2 -13744.326} C_VEL
LIN {X 0,Y 349.934,Z 190.538,A -85,B 0,C 180,E1 -13746.91,E2 -13746.91} C_VEL
LIN {X 0,Y 350.622,Z 194.244,A -85,B 0,C 180,E1 -13747.103,E2 -13747.103} C_VEL
LIN {X 0,Y 355.371,Z 218.327,A -85,B 0,C 180,E1 -13747.938,E2 -13747.938} C_VEL
LIN {X 0,Y 356.916,Z 228.053,A -85,B 0,C 180,E1 -13748.244,E2 -13748.244} C_VEL
LIN {X 0,Y 355.677,Z 295.423,A -85,B 0,C 180,E1 -13749.619,E2 -13749.619} C_VEL
LIN {X 0,Y 355.238,Z 305.301,A -85,B 0,C 180,E1 -13749.933,E2 -13749.933} C_VEL
LIN {X 0,Y 354.566,Z 315.274,A -85,B 0,C 180,E1 -13750.384,E2 -13750.384} C_VEL
LIN {X 0,Y 353.839,Z 324.629,A -85,B 0,C 180,E1 -13750.945,E2 -13750.945} C_VEL
LIN {X 0,Y 352.903,Z 334.768,A -85,B 0,C 180,E1 -13751.72,E2 -13751.72} C_VEL
LIN {X 0,Y 351.921,Z 343.762,A -85,B 0,C 180,E1 -13752.569,E2 -13752.569} C_VEL
LIN {X 0,Y 350.9,Z 352.489,A -85,B 0,C 180,E1 -13753.567,E2 -13753.567} C_VEL
LIN {X 0,Y 350.17,Z 359.04,A -85,B 0,C 180,E1 -13754.447,E2 -13754.447} C_VEL
LIN {X 0,Y 349.281,Z 367.106,A -85,B 0,C 180,E1 -13755.73,E2 -13755.73} C_VEL
LIN {X 0,Y 348.526,Z 373.308,A -85,B 0,C 180,E1 -13756.888,E2 -13756.888} C_VEL
LIN {X 0,Y 347.681,Z 379.843,A -85,B 0,C 180,E1 -13758.338,E2 -13758.338} C_VEL
LIN {X 0,Y 347.25,Z 384.347,A -85,B 0,C 180,E1 -13759.505,E2 -13759.505} C_VEL
LIN {X 0,Y 346.682,Z 389.838,A -85,B 0,C 180,E1 -13761.255,E2 -13761.255} C_VEL
LIN {X 0,Y 346.344,Z 394.163,A -85,B 0,C 180,E1 -13763.007,E2 -13763.007} C_VEL
LIN {X 0,Y 346.203,Z 396.531,A -85,B 0,C 180,E1 -13764.174,E2 -13764.174} C_VEL
LIN {X 0,Y 346.162,Z 398.331,A -85,B 0,C 180,E1 -13765.342,E2 -13765.342} C_VEL
LIN {X 0,Y 346.084,Z 400.776,A -85,B 0,C 180,E1 -13767.672,E2 -13767.672} C_VEL
LIN {X 0,Y 346.104,Z 401.365,A -85,B 0,C 180,E1 -13768.836,E2 -13768.836} C_VEL
LIN {X 0,Y 346.104,Z 401.365,A -85,B 0,C 180,E1 -13771.164,E2 -13771.164} C_VEL
LIN {X 0,Y 346.084,Z 400.776,A -85,B 0,C 180,E1 -13772.328,E2 -13772.328} C_VEL
LIN {X 0,Y 346.161,Z 398.331,A -85,B 0,C 180,E1 -13774.658,E2 -13774.658} C_VEL
LIN {X 0,Y 346.247,Z 395.381,A -85,B 0,C 180,E1 -13776.409,E2 -13776.409} C_VEL
LIN {X 0,Y 346.552,Z 391.392,A -85,B 0,C 180,E1 -13778.161,E2 -13778.161} C_VEL
LIN {X 0,Y 347.016,Z 386.262,A -85,B 0,C 180,E1 -13779.913,E2 -13779.913} C_VEL
LIN {X 0,Y 347.546,Z 380.999,A -85,B 0,C 180,E1 -13781.371,E2 -13781.371} C_VEL
LIN {X 0,Y 348.349,Z 374.683,A -85,B 0,C 180,E1 -13782.822,E2 -13782.822} C_VEL
LIN {X 0,Y 349.071,Z 368.733,A -85,B 0,C 180,E1 -13783.981,E2 -13783.981} C_VEL
LIN {X 0,Y 350.042,Z 360.694,A -85,B 0,C 180,E1 -13785.302,E2 -13785.302} C_VEL
LIN {X 0,Y 350.945,Z 352.49,A -85,B 0,C 180,E1 -13786.431,E2 -13786.431} C_VEL
LIN {X 0,Y 351.911,Z 343.762,A -85,B 0,C 180,E1 -13787.431,E2 -13787.431} C_VEL
LIN {X 0,Y 352.87,Z 334.767,A -85,B 0,C 180,E1 -13788.281,E2 -13788.281} C_VEL
LIN {X 0,Y 353.862,Z 324.629,A -85,B 0,C 180,E1 -13789.054,E2 -13789.054} C_VEL
LIN {X 0,Y 354.747,Z 312.699,A -85,B 0,C 180,E1 -13789.757,E2 -13789.757} C_VEL
LIN {X 0,Y 355.549,Z 299.402,A -85,B 0,C 180,E1 -13790.275,E2 -13790.275} C_VEL
LIN {X 0,Y 356.069,Z 278.832,A -85,B 0,C 180,E1 -13790.735,E2 -13790.735} C_VEL
LIN {X 0,Y 356.811,Z 226.983,A -85,B 0,C 180,E1 -13791.785,E2 -13791.785} C_VEL
LIN {X 0,Y 352.009,Z 200.676,A -85,B 0,C 180,E1 -13792.663,E2 -13792.663} C_VEL
LIN {X 0,Y 349.904,Z 190.931,A -85,B 0,C 180,E1 -13793.043,E2 -13793.043} C_VEL
LIN {X 0,Y 349.922,Z 189.824,A -85,B 0,C 180,E1 -13793.26,E2 -13793.26} C_VEL
LIN {X 0,Y 351.065,Z 180.769,A -85,B 0,C 180,E1 -13796.13,E2 -13796.13} C_VEL
LIN {X 0,Y 350.299,Z 175.09,A -85,B 0,C 180,E1 -13798.021,E2 -13798.021} C_VEL
LIN {X 0,Y 348.208,Z 164.53,A -85,B 0,C 180,E1 -13801.652,E2 -13801.652} C_VEL
LIN {X 0,Y 347.771,Z 162.682,A -85,B 0,C 180,E1 -13802.377,E2 -13802.377} C_VEL
LIN {X 0,Y 347.773,Z 162.652,A -85,B 0,C 180,E1 -13806.065,E2 -13806.065} C_VEL
LIN {X 0,Y 347.754,Z 162.656,A -85,B 0,C 180,E1 -13808.792,E2 -13808.792} C_VEL
LIN {X 0,Y 347.751,Z 162.655,A -85,B 0,C 180,E1 -13811.83,E2 -13811.83} C_VEL
LIN {X 0,Y 347.706,Z 162.667,A -85,B 0,C 180,E1 -13815.026,E2 -13815.026} C_VEL
LIN {X 0,Y 347.75,Z 162.665,A -85,B 0,C 180,E1 -13818.397,E2 -13818.397} C_VEL
LIN {X 0,Y 347.772,Z 162.664,A -85,B 0,C 180,E1 -13822.011,E2 -13822.011} C_VEL
LIN {X 0,Y 347.744,Z 162.65,A -85,B 0,C 180,E1 -13825.535,E2 -13825.535} C_VEL
LIN {X 0,Y 347.744,Z 162.665,A -85,B 0,C 180,E1 -13828.3,E2 -13828.3} C_VEL
LIN {X 0,Y 347.777,Z 162.657,A -85,B 0,C 180,E1 -13830.987,E2 -13830.987} C_VEL
LIN {X 0,Y 347.829,Z 162.637,A -85,B 0,C 180,E1 -13833.607,E2 -13833.607} C_VEL
LIN {X 0,Y 347.788,Z 162.658,A -85,B 0,C 180,E1 -13836.161,E2 -13836.161} C_VEL
LIN {X 0,Y 347.811,Z 162.643,A -85,B 0,C 180,E1 -13839.909,E2 -13839.909} C_VEL
LIN {X 0,Y 347.865,Z 162.629,A -85,B 0,C 180,E1 -13842.359,E2 -13842.359} C_VEL
LIN {X 0,Y 347.895,Z 162.646,A -85,B 0,C 180,E1 -13845.97,E2 -13845.97} C_VEL
LIN {X 0,Y 347.926,Z 162.619,A -85,B 0,C 180,E1 -13849.525,E2 -13849.525} C_VEL
LIN {X 0,Y 348.09,Z 162.618,A -85,B 0,C 180,E1 -13853.041,E2 -13853.041} C_VEL
LIN {X 0,Y 348.203,Z 162.603,A -85,B 0,C 180,E1 -13857.686,E2 -13857.686} C_VEL
LIN {X 0,Y 348.322,Z 162.565,A -85,B 0,C 180,E1 -13859.999,E2 -13859.999} C_VEL
LIN {X 0,Y 348.205,Z 162.595,A -85,B 0,C 180,E1 -13862.313,E2 -13862.313} C_VEL
LIN {X 0,Y 348.104,Z 162.615,A -85,B 0,C 180,E1 -13866.957,E2 -13866.957} C_VEL
LIN {X 0,Y 347.925,Z 162.618,A -85,B 0,C 180,E1 -13870.474,E2 -13870.474} C_VEL
LIN {X 0,Y 347.895,Z 162.652,A -85,B 0,C 180,E1 -13874.149,E2 -13874.149} C_VEL
LIN {X 0,Y 347.886,Z 162.624,A -85,B 0,C 180,E1 -13878.29,E2 -13878.29} C_VEL
LIN {X 0,Y 347.784,Z 162.656,A -85,B 0,C 180,E1 -13881.635,E2 -13881.635} C_VEL
LIN {X 0,Y 347.809,Z 162.657,A -85,B 0,C 180,E1 -13885.108,E2 -13885.108} C_VEL
LIN {X 0,Y 347.808,Z 162.639,A -85,B 0,C 180,E1 -13887.693,E2 -13887.693} C_VEL
LIN {X 0,Y 347.76,Z 162.666,A -85,B 0,C 180,E1 -13890.346,E2 -13890.346} C_VEL
LIN {X 0,Y 347.74,Z 162.648,A -85,B 0,C 180,E1 -13894.464,E2 -13894.464} C_VEL
LIN {X 0,Y 347.772,Z 162.665,A -85,B 0,C 180,E1 -13897.989,E2 -13897.989} C_VEL
LIN {X 0,Y 347.746,Z 162.663,A -85,B 0,C 180,E1 -13901.83,E2 -13901.83} C_VEL
LIN {X 0,Y 347.762,Z 162.656,A -85,B 0,C 180,E1 -13905.016,E2 -13905.016} C_VEL
LIN {X 0,Y 347.745,Z 162.623,A -85,B 0,C 180,E1 -13908.397,E2 -13908.397} C_VEL
LIN {X 0,Y 347.772,Z 162.665,A -85,B 0,C 180,E1 -13912.01,E2 -13912.01} C_VEL
LIN {X 0,Y 347.74,Z 162.641,A -85,B 0,C 180,E1 -13915.536,E2 -13915.536} C_VEL
LIN {X 0,Y 347.762,Z 162.668,A -85,B 0,C 180,E1 -13918.303,E2 -13918.303} C_VEL
LIN {X 0,Y 347.802,Z 162.643,A -85,B 0,C 180,E1 -13920.99,E2 -13920.99} C_VEL
LIN {X 0,Y 347.828,Z 162.66,A -85,B 0,C 180,E1 -13923.608,E2 -13923.608} C_VEL
LIN {X 0,Y 347.784,Z 162.666,A -85,B 0,C 180,E1 -13926.162,E2 -13926.162} C_VEL
LIN {X 0,Y 347.821,Z 162.782,A -85,B 0,C 180,E1 -13929.138,E2 -13929.138} C_VEL
LIN {X 0,Y 348.019,Z 163.798,A -85,B 0,C 180,E1 -13929.459,E2 -13929.459} C_VEL
LIN {X 0,Y 349.6,Z 166.556,A -85,B 0,C 180,E1 -13929.906,E2 -13929.906} C_VEL
LIN {X 0,Y 351.805,Z 168.417,A -85,B 0,C 180,E1 -13930.407,E2 -13930.407} C_VEL
LIN {X 0,Y 353.932,Z 171.744,A -85,B 0,C 180,E1 -13930.994,E2 -13930.994} C_VEL
LIN {X 0,Y 356.535,Z 174.128,A -85,B 0,C 180,E1 -13931.644,E2 -13931.644} C_VEL
LIN {X 0,Y 359.05,Z 177.504,A -85,B 0,C 180,E1 -13932.356,E2 -13932.356} C_VEL
LIN {X 0,Y 361.877,Z 180.013,A -85,B 0,C 180,E1 -13933.127,E2 -13933.127} C_VEL
LIN {X 0,Y 364.51,Z 183.267,A -85,B 0,C 180,E1 -13933.938,E2 -13933.938} C_VEL
LIN {X 0,Y 368.012,Z 186.185,A -85,B 0,C 180,E1 -13934.996,E2 -13934.996} C_VEL
LIN {X 0,Y 370.998,Z 189.698,A -85,B 0,C 180,E1 -13936.035,E2 -13936.035} C_VEL
LIN {X 0,Y 374.573,Z 192.558,A -85,B 0,C 180,E1 -13937.329,E2 -13937.329} C_VEL
LIN {X 0,Y 377.47,Z 195.84,A -85,B 0,C 180,E1 -13938.533,E2 -13938.533} C_VEL
LIN {X 0,Y 380.315,Z 198.007,A -85,B 0,C 180,E1 -13939.787,E2 -13939.787} C_VEL
LIN {X 0,Y 382.425,Z 199.252,A -85,B 0,C 180,E1 -13940.794,E2 -13940.794} C_VEL
LIN {X 0,Y 385.153,Z 202.561,A -85,B 0,C 180,E1 -13942.452,E2 -13942.452} C_VEL
LIN {X 0,Y 387.586,Z 204.46,A -85,B 0,C 180,E1 -13944.251,E2 -13944.251} C_VEL
LIN {X 0,Y 389.26,Z 205.376,A -85,B 0,C 180,E1 -13945.859,E2 -13945.859} C_VEL
LIN {X 0,Y 390.395,Z 205.749,A -85,B 0,C 180,E1 -13947.439,E2 -13947.439} C_VEL
LIN {X 0,Y 390.961,Z 206.178,A -85,B 0,C 180,E1 -13948.97,E2 -13948.97} C_VEL
LIN {X 0,Y 391.134,Z 206.115,A -85,B 0,C 180,E1 -13950,E2 -13950} C_VEL
LIN {X 0,Y 390.861,Z 206.065,A -85,B 0,C 180,E1 -13951.546,E2 -13951.546} C_VEL
LIN {X 0,Y 390.115,Z 205.607,A -85,B 0,C 180,E1 -13953.098,E2 -13953.098} C_VEL
LIN {X 0,Y 388.503,Z 205.027,A -85,B 0,C 180,E1 -13954.929,E2 -13954.929} C_VEL
LIN {X 0,Y 386.387,Z 203.614,A -85,B 0,C 180,E1 -13956.668,E2 -13956.668} C_VEL
LIN {X 0,Y 384.293,Z 201.698,A -85,B 0,C 180,E1 -13958.072,E2 -13958.072} C_VEL
LIN {X 0,Y 382.054,Z 198.875,A -85,B 0,C 180,E1 -13959.396,E2 -13959.396} C_VEL
LIN {X 0,Y 378.834,Z 196.988,A -85,B 0,C 180,E1 -13960.894,E2 -13960.894} C_VEL
LIN {X 0,Y 375.359,Z 193.576,A -85,B 0,C 180,E1 -13962.365,E2 -13962.365} C_VEL
LIN {X 0,Y 373.857,Z 191.856,A -85,B 0,C 180,E1 -13962.942,E2 -13962.942} C_VEL
LIN {X 0,Y 370.642,Z 189.352,A -85,B 0,C 180,E1 -13964.084,E2 -13964.084} C_VEL
LIN {X 0,Y 367.17,Z 185.335,A -85,B 0,C 180,E1 -13965.274,E2 -13965.274} C_VEL
LIN {X 0,Y 363.714,Z 182.426,A -85,B 0,C 180,E1 -13966.311,E2 -13966.311} C_VEL
LIN {X 0,Y 360.955,Z 179.101,A -85,B 0,C 180,E1 -13967.125,E2 -13967.125} C_VEL
LIN {X 0,Y 358.145,Z 176.488,A -85,B 0,C 180,E1 -13967.904,E2 -13967.904} C_VEL
LIN {X 0,Y 356.111,Z 173.541,A -85,B 0,C 180,E1 -13968.467,E2 -13968.467} C_VEL
LIN {X 0,Y 353.385,Z 171.09,A -85,B 0,C 180,E1 -13969.15,E2 -13969.15} C_VEL
LIN {X 0,Y 351.55,Z 168.059,A -85,B 0,C 180,E1 -13969.659,E2 -13969.659} C_VEL
LIN {X 0,Y 349.254,Z 166.179,A -85,B 0,C 180,E1 -13970.175,E2 -13970.175} C_VEL
LIN {X 0,Y 347.917,Z 163.336,A -85,B 0,C 180,E1 -13970.624,E2 -13970.624} C_VEL
LIN {X 0,Y 347.811,Z 162.699,A -85,B 0,C 180,E1 -13971.018,E2 -13971.018} C_VEL
LIN {X 0,Y 347.808,Z 162.662,A -85,B 0,C 180,E1 -13975.108,E2 -13975.108} C_VEL
LIN {X 0,Y 347.808,Z 162.658,A -85,B 0,C 180,E1 -13977.694,E2 -13977.694} C_VEL
LIN {X 0,Y 347.767,Z 162.654,A -85,B 0,C 180,E1 -13980.346,E2 -13980.346} C_VEL
LIN {X 0,Y 347.744,Z 162.642,A -85,B 0,C 180,E1 -13984.044,E2 -13984.044} C_VEL
LIN {X 0,Y 347.761,Z 162.667,A -85,B 0,C 180,E1 -13987.32,E2 -13987.32} C_VEL
LIN {X 0,Y 347.727,Z 162.644,A -85,B 0,C 180,E1 -13990.297,E2 -13990.297} C_VEL
LIN {X 0,Y 347.721,Z 162.637,A -85,B 0,C 180,E1 -13993.408,E2 -13993.408} C_VEL
LIN {X 0,Y 347.723,Z 162.674,A -85,B 0,C 180,E1 -13996.686,E2 -13996.686} C_VEL
LIN {X 0,Y 347.742,Z 162.657,A -85,B 0,C 180,E1 -14000.173,E2 -14000.173} C_VEL
LIN {X 0,Y 347.761,Z 162.668,A -85,B 0,C 180,E1 -14002.68,E2 -14002.68} C_VEL
LIN {X 0,Y 347.743,Z 162.649,A -85,B 0,C 180,E1 -14005.957,E2 -14005.957} C_VEL
LIN {X 0,Y 347.751,Z 162.666,A -85,B 0,C 180,E1 -14009.541,E2 -14009.541} C_VEL
LIN {X 0,Y 347.143,Z 162.744,A -85,B 0,C 180,E1 -14010.509,E2 -14010.509} C_VEL
LIN {X 0,Y 344.321,Z 163.088,A -85,B 0,C 180,E1 -14012.083,E2 -14012.083} C_VEL
LIN {X 0,Y 341.892,Z 163.383,A -85,B 0,C 180,E1 -14013.358,E2 -14013.358} C_VEL
LIN {X 0,Y 340.844,Z 163.515,A -85,B 0,C 180,E1 -14014.344,E2 -14014.344} C_VEL
LIN {X 0,Y 340.757,Z 163.528,A -85,B 0,C 180,E1 -14014.679,E2 -14014.679} C_VEL
LIN {X 0,Y 340.737,Z 163.535,A -85,B 0,C 180,E1 -14018.207,E2 -14018.207} C_VEL
LIN {X 0,Y 340.853,Z 163.502,A -85,B 0,C 180,E1 -14021.985,E2 -14021.985} C_VEL
LIN {X 0,Y 340.866,Z 163.526,A -85,B 0,C 180,E1 -14025.706,E2 -14025.706} C_VEL
LIN {X 0,Y 340.867,Z 163.498,A -85,B 0,C 180,E1 -14029.307,E2 -14029.307} C_VEL
LIN {X 0,Y 341.074,Z 163.491,A -85,B 0,C 180,E1 -14032.899,E2 -14032.899} C_VEL
LIN {X 0,Y 341.167,Z 163.472,A -85,B 0,C 180,E1 -14037.639,E2 -14037.639} C_VEL
LIN {X 0,Y 341.272,Z 163.442,A -85,B 0,C 180,E1 -14040.001,E2 -14040.001} C_VEL
LIN {X 0,Y 341.165,Z 163.479,A -85,B 0,C 180,E1 -14042.362,E2 -14042.362} C_VEL
LIN {X 0,Y 341.058,Z 163.491,A -85,B 0,C 180,E1 -14047.103,E2 -14047.103} C_VEL
LIN {X 0,Y 340.868,Z 163.498,A -85,B 0,C 180,E1 -14050.694,E2 -14050.694} C_VEL
LIN {X 0,Y 340.861,Z 163.522,A -85,B 0,C 180,E1 -14054.326,E2 -14054.326} C_VEL
LIN {X 0,Y 340.835,Z 163.499,A -85,B 0,C 180,E1 -14058.467,E2 -14058.467} C_VEL
LIN {X 0,Y 340.752,Z 163.535,A -85,B 0,C 180,E1 -14061.858,E2 -14061.858} C_VEL
LIN {X 0,Y 340.771,Z 163.52,A -85,B 0,C 180,E1 -14065.665,E2 -14065.665} C_VEL
LIN {X 0,Y 340.727,Z 163.527,A -85,B 0,C 180,E1 -14068.322,E2 -14068.322} C_VEL
LIN {X 0,Y 340.697,Z 163.546,A -85,B 0,C 180,E1 -14071.045,E2 -14071.045} C_VEL
LIN {X 0,Y 340.717,Z 163.533,A -85,B 0,C 180,E1 -14075.28,E2 -14075.28} C_VEL
LIN {X 0,Y 340.709,Z 163.543,A -85,B 0,C 180,E1 -14078.387,E2 -14078.387} C_VEL
LIN {X 0,Y 340.699,Z 163.544,A -85,B 0,C 180,E1 -14082.046,E2 -14082.046} C_VEL
LIN {X 0,Y 340.652,Z 163.553,A -85,B 0,C 180,E1 -14086.228,E2 -14086.228} C_VEL
LIN {X 0,Y 340.688,Z 163.522,A -85,B 0,C 180,E1 -14089.754,E2 -14089.754} C_VEL
LIN {X 0,Y 340.708,Z 163.539,A -85,B 0,C 180,E1 -14093.259,E2 -14093.259} C_VEL
LIN {X 0,Y 340.713,Z 163.54,A -85,B 0,C 180,E1 -14096.865,E2 -14096.865} C_VEL
LIN {X 0,Y 340.787,Z 163.857,A -85,B 0,C 180,E1 -14097.4,E2 -14097.4} C_VEL
LIN {X 0,Y 342.288,Z 171.092,A -85,B 0,C 180,E1 -14100.081,E2 -14100.081} C_VEL
LIN {X 0,Y 343.749,Z 178.595,A -85,B 0,C 180,E1 -14102.612,E2 -14102.612} C_VEL
LIN {X 0,Y 344.006,Z 182.753,A -85,B 0,C 180,E1 -14104.017,E2 -14104.017} C_VEL
LIN {X 0,Y 343.054,Z 190.277,A -85,B 0,C 180,E1 -14106.406,E2 -14106.406} C_VEL
LIN {X 0,Y 343.386,Z 192.379,A -85,B 0,C 180,E1 -14106.556,E2 -14106.556} C_VEL
LIN {X 0,Y 348.56,Z 217.719,A -85,B 0,C 180,E1 -14107.475,E2 -14107.475} C_VEL
LIN {X 0,Y 350.344,Z 229.03,A -85,B 0,C 180,E1 -14107.84,E2 -14107.84} C_VEL
LIN {X 0,Y 349.041,Z 295.238,A -85,B 0,C 180,E1 -14109.214,E2 -14109.214} C_VEL
LIN {X 0,Y 348.591,Z 305.11,A -85,B 0,C 180,E1 -14109.533,E2 -14109.533} C_VEL
LIN {X 0,Y 347.9,Z 315.083,A -85,B 0,C 180,E1 -14109.992,E2 -14109.992} C_VEL
LIN {X 0,Y 347.137,Z 324.437,A -85,B 0,C 180,E1 -14110.562,E2 -14110.562} C_VEL
LIN {X 0,Y 346.157,Z 334.576,A -85,B 0,C 180,E1 -14111.351,E2 -14111.351} C_VEL
LIN {X 0,Y 345.124,Z 343.57,A -85,B 0,C 180,E1 -14112.215,E2 -14112.215} C_VEL
LIN {X 0,Y 344.079,Z 352.297,A -85,B 0,C 180,E1 -14113.231,E2 -14113.231} C_VEL
LIN {X 0,Y 343.19,Z 359.705,A -85,B 0,C 180,E1 -14114.258,E2 -14114.258} C_VEL
LIN {X 0,Y 342.346,Z 366.913,A -85,B 0,C 180,E1 -14115.435,E2 -14115.435} C_VEL
LIN {X 0,Y 341.591,Z 373.115,A -85,B 0,C 180,E1 -14116.617,E2 -14116.617} C_VEL
LIN {X 0,Y 340.708,Z 379.651,A -85,B 0,C 180,E1 -14118.096,E2 -14118.096} C_VEL
LIN {X 0,Y 340.235,Z 384.154,A -85,B 0,C 180,E1 -14119.286,E2 -14119.286} C_VEL
LIN {X 0,Y 339.654,Z 389.646,A -85,B 0,C 180,E1 -14121.072,E2 -14121.072} C_VEL
LIN {X 0,Y 339.275,Z 393.971,A -85,B 0,C 180,E1 -14122.86,E2 -14122.86} C_VEL
LIN {X 0,Y 339.134,Z 396.436,A -85,B 0,C 180,E1 -14124.116,E2 -14124.116} C_VEL
LIN {X 0,Y 339.067,Z 399.527,A -85,B 0,C 180,E1 -14126.435,E2 -14126.435} C_VEL
LIN {X 0,Y 338.998,Z 400.584,A -85,B 0,C 180,E1 -14127.624,E2 -14127.624} C_VEL
LIN {X 0,Y 339.007,Z 401.174,A -85,B 0,C 180,E1 -14128.812,E2 -14128.812} C_VEL
LIN {X 0,Y 339.007,Z 401.174,A -85,B 0,C 180,E1 -14131.188,E2 -14131.188} C_VEL
LIN {X 0,Y 338.998,Z 400.584,A -85,B 0,C 180,E1 -14132.376,E2 -14132.376} C_VEL
LIN {X 0,Y 339.063,Z 398.138,A -85,B 0,C 180,E1 -14134.756,E2 -14134.756} C_VEL
LIN {X 0,Y 339.17,Z 395.188,A -85,B 0,C 180,E1 -14136.544,E2 -14136.544} C_VEL
LIN {X 0,Y 339.511,Z 391.2,A -85,B 0,C 180,E1 -14138.332,E2 -14138.332} C_VEL
LIN {X 0,Y 339.992,Z 386.069,A -85,B 0,C 180,E1 -14140.12,E2 -14140.12} C_VEL
LIN {X 0,Y 340.556,Z 380.806,A -85,B 0,C 180,E1 -14141.608,E2 -14141.608} C_VEL
LIN {X 0,Y 341.403,Z 374.491,A -85,B 0,C 180,E1 -14143.088,E2 -14143.088} C_VEL
LIN {X 0,Y 342.137,Z 368.54,A -85,B 0,C 180,E1 -14144.27,E2 -14144.27} C_VEL
LIN {X 0,Y 343.139,Z 360.597,A -85,B 0,C 180,E1 -14145.603,E2 -14145.603} C_VEL
LIN {X 0,Y 343.981,Z 353.433,A -85,B 0,C 180,E1 -14146.621,E2 -14146.621} C_VEL
LIN {X 0,Y 344.981,Z 344.922,A -85,B 0,C 180,E1 -14147.64,E2 -14147.64} C_VEL
LIN {X 0,Y 345.958,Z 336.207,A -85,B 0,C 180,E1 -14148.506,E2 -14148.506} C_VEL
LIN {X 0,Y 346.97,Z 326.452,A -85,B 0,C 180,E1 -14149.294,E2 -14149.294} C_VEL
LIN {X 0,Y 347.779,Z 316.37,A -85,B 0,C 180,E1 -14149.938,E2 -14149.938} C_VEL
LIN {X 0,Y 348.452,Z 306.857,A -85,B 0,C 180,E1 -14150.398,E2 -14150.398} C_VEL
LIN {X 0,Y 349.007,Z 296.548,A -85,B 0,C 180,E1 -14150.75,E2 -14150.75} C_VEL
LIN {X 0,Y 350.277,Z 229.378,A -85,B 0,C 180,E1 -14152.157,E2 -14152.157} C_VEL
LIN {X 0,Y 348.619,Z 218.394,A -85,B 0,C 180,E1 -14152.507,E2 -14152.507} C_VEL
LIN {X 0,Y 344.028,Z 195.227,A -85,B 0,C 180,E1 -14153.335,E2 -14153.335} C_VEL
LIN {X 0,Y 343.052,Z 190.601,A -85,B 0,C 180,E1 -14153.543,E2 -14153.543} C_VEL
LIN {X 0,Y 343.262,Z 188.343,A -85,B 0,C 180,E1 -14154.172,E2 -14154.172} C_VEL
LIN {X 0,Y 344.104,Z 181.869,A -85,B 0,C 180,E1 -14156.269,E2 -14156.269} C_VEL
LIN {X 0,Y 343.253,Z 175.927,A -85,B 0,C 180,E1 -14158.307,E2 -14158.307} C_VEL
LIN {X 0,Y 341.391,Z 166.556,A -85,B 0,C 180,E1 -14161.618,E2 -14161.618} C_VEL
LIN {X 0,Y 340.728,Z 163.555,A -85,B 0,C 180,E1 -14162.782,E2 -14162.782} C_VEL
LIN {X 0,Y 340.713,Z 163.535,A -85,B 0,C 180,E1 -14166.44,E2 -14166.44} C_VEL
LIN {X 0,Y 340.7,Z 163.522,A -85,B 0,C 180,E1 -14169.752,E2 -14169.752} C_VEL
LIN {X 0,Y 340.676,Z 163.548,A -85,B 0,C 180,E1 -14172.904,E2 -14172.904} C_VEL
LIN {X 0,Y 340.676,Z 163.549,A -85,B 0,C 180,E1 -14177.095,E2 -14177.095} C_VEL
LIN {X 0,Y 340.699,Z 163.534,A -85,B 0,C 180,E1 -14180.247,E2 -14180.247} C_VEL
LIN {X 0,Y 340.709,Z 163.541,A -85,B 0,C 180,E1 -14183.559,E2 -14183.559} C_VEL
LIN {X 0,Y 340.691,Z 163.528,A -85,B 0,C 180,E1 -14186.153,E2 -14186.153} C_VEL
LIN {X 0,Y 340.74,Z 163.538,A -85,B 0,C 180,E1 -14190.329,E2 -14190.329} C_VEL
LIN {X 0,Y 340.802,Z 163.51,A -85,B 0,C 180,E1 -14193.019,E2 -14193.019} C_VEL
LIN {X 0,Y 340.728,Z 163.543,A -85,B 0,C 180,E1 -14196.926,E2 -14196.926} C_VEL
LIN {X 0,Y 340.789,Z 163.507,A -85,B 0,C 180,E1 -14200.733,E2 -14200.733} C_VEL
LIN {X 0,Y 340.785,Z 163.52,A -85,B 0,C 180,E1 -14203.218,E2 -14203.218} C_VEL
LIN {X 0,Y 340.842,Z 163.522,A -85,B 0,C 180,E1 -14206.89,E2 -14206.89} C_VEL
LIN {X 0,Y 340.911,Z 163.487,A -85,B 0,C 180,E1 -14210.507,E2 -14210.507} C_VEL
LIN {X 0,Y 341.058,Z 163.491,A -85,B 0,C 180,E1 -14212.897,E2 -14212.897} C_VEL
LIN {X 0,Y 341.165,Z 163.479,A -85,B 0,C 180,E1 -14217.638,E2 -14217.638} C_VEL
LIN {X 0,Y 341.272,Z 163.442,A -85,B 0,C 180,E1 -14219.999,E2 -14219.999} C_VEL
LIN {X 0,Y 341.167,Z 163.472,A -85,B 0,C 180,E1 -14222.361,E2 -14222.361} C_VEL
LIN {X 0,Y 341.074,Z 163.491,A -85,B 0,C 180,E1 -14227.101,E2 -14227.101} C_VEL
LIN {X 0,Y 340.867,Z 163.498,A -85,B 0,C 180,E1 -14230.693,E2 -14230.693} C_VEL
LIN {X 0,Y 340.859,Z 163.527,A -85,B 0,C 180,E1 -14234.324,E2 -14234.324} C_VEL
LIN {X 0,Y 340.833,Z 163.501,A -85,B 0,C 180,E1 -14238.466,E2 -14238.466} C_VEL
LIN {X 0,Y 340.75,Z 163.534,A -85,B 0,C 180,E1 -14241.856,E2 -14241.856} C_VEL
LIN {X 0,Y 340.769,Z 163.524,A -85,B 0,C 180,E1 -14245.664,E2 -14245.664} C_VEL
LIN {X 0,Y 340.738,Z 163.525,A -85,B 0,C 180,E1 -14248.319,E2 -14248.319} C_VEL
